LIN {X 0,Y 311.231,Z 437.384,A -85,B 0,C 180,E1 -15755.184,E2 -15755.184} C_VEL
LIN {X 0,Y 311.07,Z 439.493,A -85,B 0,C 180,E1 -15756.488,E2 -15756.488} C_VEL
LIN {X 0,Y 310.876,Z 441.171,A -85,B 0,C 180,E1 -15757.797,E2 -15757.797} C_VEL
LIN {X 0,Y 310.751,Z 442.446,A -85,B 0,C 180,E1 -15759.111,E2 -15759.111} C_VEL
LIN {X 0,Y 310.679,Z 443.314,A -85,B 0,C 180,E1 -15760.428,E2 -15760.428} C_VEL
LIN {X 0,Y 310.751,Z 443.737,A -85,B 0,C 180,E1 -15761.746,E2 -15761.746} C_VEL
LIN {X 0,Y 310.874,Z 443.708,A -85,B 0,C 180,E1 -15763.562,E2 -15763.562} C_VEL
LIN {X 0,Y 311.133,Z 442.642,A -85,B 0,C 180,E1 -15765.728,E2 -15765.728} C_VEL
LIN {X 0,Y 311.417,Z 441.418,A -85,B 0,C 180,E1 -15767.061,E2 -15767.061} C_VEL
LIN {X 0,Y 312.024,Z 439.019,A -85,B 0,C 180,E1 -15768.913,E2 -15768.913} C_VEL
LIN {X 0,Y 312.86,Z 435.083,A -85,B 0,C 180,E1 -15771.065,E2 -15771.065} C_VEL
LIN {X 0,Y 313.883,Z 430.519,A -85,B 0,C 180,E1 -15772.948,E2 -15772.948} C_VEL
LIN {X 0,Y 315.274,Z 423.973,A -85,B 0,C 180,E1 -15775.058,E2 -15775.058} C_VEL
LIN {X 0,Y 316.969,Z 416.151,A -85,B 0,C 180,E1 -15777.035,E2 -15777.035} C_VEL
LIN {X 0,Y 318.681,Z 407.222,A -85,B 0,C 180,E1 -15778.825,E2 -15778.825} C_VEL
LIN {X 0,Y 320.497,Z 396.978,A -85,B 0,C 180,E1 -15780.47,E2 -15780.47} C_VEL
LIN {X 0,Y 322.265,Z 386.498,A -85,B 0,C 180,E1 -15781.793,E2 -15781.793} C_VEL
LIN {X 0,Y 323.658,Z 375.789,A -85,B 0,C 180,E1 -15782.877,E2 -15782.877} C_VEL
LIN {X 0,Y 324.815,Z 364.59,A -85,B 0,C 180,E1 -15783.765,E2 -15783.765} C_VEL
LIN {X 0,Y 325.961,Z 351.288,A -85,B 0,C 180,E1 -15784.526,E2 -15784.526} C_VEL
LIN {X 0,Y 326.606,Z 338.938,A -85,B 0,C 180,E1 -15784.984,E2 -15784.984} C_VEL
LIN {X 0,Y 328.652,Z 266.261,A -85,B 0,C 180,E1 -15786.6,E2 -15786.6} C_VEL
LIN {X 0,Y 321.5,Z 250.026,A -85,B 0,C 180,E1 -15787.749,E2 -15787.749} C_VEL
LIN {X 0,Y 314.331,Z 235.95,A -85,B 0,C 180,E1 -15788.911,E2 -15788.911} C_VEL
LIN {X 0,Y 314.024,Z 235.367,A -85,B 0,C 180,E1 -15788.962,E2 -15788.962} C_VEL
LIN {X 0,Y 312.775,Z 233.899,A -85,B 0,C 180,E1 -15789.216,E2 -15789.216} C_VEL
LIN {X 0,Y 309.925,Z 232.398,A -85,B 0,C 180,E1 -15789.967,E2 -15789.967} C_VEL
LIN {X 0,Y 308.287,Z 231.569,A -85,B 0,C 180,E1 -15790.527,E2 -15790.527} C_VEL
LIN {X 0,Y 306.002,Z 231.431,A -85,B 0,C 180,E1 -15791.683,E2 -15791.683} C_VEL
LIN {X 0,Y 305.488,Z 231.435,A -85,B 0,C 180,E1 -15792.497,E2 -15792.497} C_VEL
LIN {X 0,Y 305.487,Z 231.436,A -85,B 0,C 180,E1 -15796.356,E2 -15796.356} C_VEL
LIN {X 0,Y 305.476,Z 231.431,A -85,B 0,C 180,E1 -15799.895,E2 -15799.895} C_VEL
LIN {X 0,Y 305.474,Z 231.432,A -85,B 0,C 180,E1 -15803.63,E2 -15803.63} C_VEL
LIN {X 0,Y 305.455,Z 231.435,A -85,B 0,C 180,E1 -15806.482,E2 -15806.482} C_VEL
LIN {X 0,Y 305.483,Z 231.432,A -85,B 0,C 180,E1 -15810.95,E2 -15810.95} C_VEL
LIN {X 0,Y 305.557,Z 231.425,A -85,B 0,C 180,E1 -15814.086,E2 -15814.086} C_VEL
LIN {X 0,Y 305.449,Z 231.436,A -85,B 0,C 180,E1 -15818.399,E2 -15818.399} C_VEL
LIN {X 0,Y 305.531,Z 231.419,A -85,B 0,C 180,E1 -15821.214,E2 -15821.214} C_VEL
LIN {X 0,Y 305.608,Z 231.409,A -85,B 0,C 180,E1 -15825.347,E2 -15825.347} C_VEL
LIN {X 0,Y 305.608,Z 231.409,A -85,B 0,C 180,E1 -15829.398,E2 -15829.398} C_VEL
LIN {X 0,Y 305.769,Z 231.395,A -85,B 0,C 180,E1 -15832.073,E2 -15832.073} C_VEL
LIN {X 0,Y 305.662,Z 231.404,A -85,B 0,C 180,E1 -15834.723,E2 -15834.723} C_VEL
LIN {X 0,Y 305.934,Z 231.365,A -85,B 0,C 180,E1 -15838.684,E2 -15838.684} C_VEL
LIN {X 0,Y 305.934,Z 231.375,A -85,B 0,C 180,E1 -15841.316,E2 -15841.316} C_VEL
LIN {X 0,Y 305.648,Z 231.413,A -85,B 0,C 180,E1 -15845.277,E2 -15845.277} C_VEL
LIN {X 0,Y 305.722,Z 231.391,A -85,B 0,C 180,E1 -15847.928,E2 -15847.928} C_VEL
LIN {X 0,Y 305.578,Z 231.412,A -85,B 0,C 180,E1 -15851.946,E2 -15851.946} C_VEL
LIN {X 0,Y 305.591,Z 231.419,A -85,B 0,C 180,E1 -15855.013,E2 -15855.013} C_VEL
LIN {X 0,Y 305.499,Z 231.43,A -85,B 0,C 180,E1 -15858.788,E2 -15858.788} C_VEL
LIN {X 0,Y 305.442,Z 231.438,A -85,B 0,C 180,E1 -15863.027,E2 -15863.027} C_VEL
LIN {X 0,Y 305.438,Z 231.429,A -85,B 0,C 180,E1 -15866.191,E2 -15866.191} C_VEL
LIN {X 0,Y 305.409,Z 231.435,A -85,B 0,C 180,E1 -15869.026,E2 -15869.026} C_VEL
LIN {X 0,Y 305.421,Z 231.44,A -85,B 0,C 180,E1 -15871.955,E2 -15871.955} C_VEL
LIN {X 0,Y 305.449,Z 231.436,A -85,B 0,C 180,E1 -15875.115,E2 -15875.115} C_VEL
LIN {X 0,Y 305.415,Z 231.415,A -85,B 0,C 180,E1 -15878.524,E2 -15878.524} C_VEL
LIN {X 0,Y 305.419,Z 231.442,A -85,B 0,C 180,E1 -15881.861,E2 -15881.861} C_VEL
LIN {X 0,Y 305.392,Z 231.441,A -85,B 0,C 180,E1 -15885.513,E2 -15885.513} C_VEL
LIN {X 0,Y 305.406,Z 231.431,A -85,B 0,C 180,E1 -15888.139,E2 -15888.139} C_VEL
LIN {X 0,Y 305.467,Z 231.429,A -85,B 0,C 180,E1 -15892.434,E2 -15892.434} C_VEL
LIN {X 0,Y 305.527,Z 231.652,A -85,B 0,C 180,E1 -15893.269,E2 -15893.269} C_VEL
LIN {X 0,Y 307.663,Z 239.802,A -85,B 0,C 180,E1 -15896.065,E2 -15896.065} C_VEL
LIN {X 0,Y 310.119,Z 250.307,A -85,B 0,C 180,E1 -15899.448,E2 -15899.448} C_VEL
LIN {X 0,Y 311.704,Z 257.977,A -85,B 0,C 180,E1 -15901.784,E2 -15901.784} C_VEL
LIN {X 0,Y 313.869,Z 263.63,A -85,B 0,C 180,E1 -15902.185,E2 -15902.185} C_VEL
LIN {X 0,Y 318.647,Z 287.185,A -85,B 0,C 180,E1 -15903.318,E2 -15903.318} C_VEL
LIN {X 0,Y 321.489,Z 305.27,A -85,B 0,C 180,E1 -15904.074,E2 -15904.074} C_VEL
LIN {X 0,Y 319.685,Z 367.009,A -85,B 0,C 180,E1 -15905.484,E2 -15905.484} C_VEL
LIN {X 0,Y 318.677,Z 380.224,A -85,B 0,C 180,E1 -15906.008,E2 -15906.008} C_VEL
LIN {X 0,Y 317.293,Z 392.914,A -85,B 0,C 180,E1 -15906.762,E2 -15906.762} C_VEL
LIN {X 0,Y 315.566,Z 405.023,A -85,B 0,C 180,E1 -15907.752,E2 -15907.752} C_VEL
LIN {X 0,Y 313.569,Z 416.536,A -85,B 0,C 180,E1 -15908.985,E2 -15908.985} C_VEL
LIN {X 0,Y 311.699,Z 426.916,A -85,B 0,C 180,E1 -15910.403,E2 -15910.403} C_VEL
LIN {X 0,Y 310.015,Z 435.426,A -85,B 0,C 180,E1 -15911.837,E2 -15911.837} C_VEL
LIN {X 0,Y 308.316,Z 443.862,A -85,B 0,C 180,E1 -15913.578,E2 -15913.578} C_VEL
LIN {X 0,Y 306.923,Z 451.023,A -85,B 0,C 180,E1 -15915.41,E2 -15915.41} C_VEL
LIN {X 0,Y 305.546,Z 457.248,A -85,B 0,C 180,E1 -15917.377,E2 -15917.377} C_VEL
LIN {X 0,Y 304.657,Z 462.223,A -85,B 0,C 180,E1 -15919.364,E2 -15919.364} C_VEL
LIN {X 0,Y 304.066,Z 466.09,A -85,B 0,C 180,E1 -15921.358,E2 -15921.358} C_VEL
LIN {X 0,Y 303.742,Z 468.951,A -85,B 0,C 180,E1 -15923.355,E2 -15923.355} C_VEL
LIN {X 0,Y 303.66,Z 471.296,A -85,B 0,C 180,E1 -15926.016,E2 -15926.016} C_VEL
LIN {X 0,Y 303.656,Z 471.885,A -85,B 0,C 180,E1 -15927.345,E2 -15927.345} C_VEL
LIN {X 0,Y 303.684,Z 472.046,A -85,B 0,C 180,E1 -15928.672,E2 -15928.672} C_VEL
LIN {X 0,Y 303.768,Z 471.804,A -85,B 0,C 180,E1 -15929.998,E2 -15929.998} C_VEL
LIN {X 0,Y 303.723,Z 471.166,A -85,B 0,C 180,E1 -15931.323,E2 -15931.323} C_VEL
LIN {X 0,Y 303.69,Z 470.133,A -85,B 0,C 180,E1 -15932.65,E2 -15932.65} C_VEL
LIN {X 0,Y 303.713,Z 468.654,A -85,B 0,C 180,E1 -15933.978,E2 -15933.978} C_VEL
LIN {X 0,Y 303.728,Z 466.023,A -85,B 0,C 180,E1 -15935.741,E2 -15935.741} C_VEL
LIN {X 0,Y 303.929,Z 461.501,A -85,B 0,C 180,E1 -15937.972,E2 -15937.972} C_VEL
LIN {X 0,Y 304.387,Z 455.17,A -85,B 0,C 180,E1 -15940.304,E2 -15940.304} C_VEL
LIN {X 0,Y 305.062,Z 448.265,A -85,B 0,C 180,E1 -15942.3,E2 -15942.3} C_VEL
LIN {X 0,Y 305.872,Z 441.212,A -85,B 0,C 180,E1 -15943.957,E2 -15943.957} C_VEL
LIN {X 0,Y 306.784,Z 433.425,A -85,B 0,C 180,E1 -15945.476,E2 -15945.476} C_VEL
LIN {X 0,Y 307.98,Z 423.495,A -85,B 0,C 180,E1 -15947.064,E2 -15947.064} C_VEL
LIN {X 0,Y 309.143,Z 413.209,A -85,B 0,C 180,E1 -15948.382,E2 -15948.382} C_VEL
LIN {X 0,Y 310.372,Z 402.142,A -85,B 0,C 180,E1 -15949.507,E2 -15949.507} C_VEL
LIN {X 0,Y 311.519,Z 389.878,A -85,B 0,C 180,E1 -15950.463,E2 -15950.463} C_VEL
LIN {X 0,Y 312.452,Z 377.055,A -85,B 0,C 180,E1 -15951.175,E2 -15951.175} C_VEL
LIN {X 0,Y 313.089,Z 363.48,A -85,B 0,C 180,E1 -15951.648,E2 -15951.648} C_VEL
LIN {X 0,Y 314.139,Z 301.472,A -85,B 0,C 180,E1 -15953.065,E2 -15953.065} C_VEL
LIN {X 0,Y 308.599,Z 258.926,A -85,B 0,C 180,E1 -15954.459,E2 -15954.459} C_VEL
LIN {X 0,Y 309.401,Z 251.713,A -85,B 0,C 180,E1 -15956.286,E2 -15956.286} C_VEL
LIN {X 0,Y 308.464,Z 245.706,A -85,B 0,C 180,E1 -15957.927,E2 -15957.927} C_VEL
LIN {X 0,Y 306.146,Z 234.57,A -85,B 0,C 180,E1 -15961.093,E2 -15961.093} C_VEL
LIN {X 0,Y 305.45,Z 231.442,A -85,B 0,C 180,E1 -15962.042,E2 -15962.042} C_VEL
LIN {X 0,Y 305.444,Z 231.437,A -85,B 0,C 180,E1 -15965.109,E2 -15965.109} C_VEL
LIN {X 0,Y 305.446,Z 231.437,A -85,B 0,C 180,E1 -15968.528,E2 -15968.528} C_VEL
LIN {X 0,Y 305.436,Z 231.437,A -85,B 0,C 180,E1 -15972.582,E2 -15972.582} C_VEL
LIN {X 0,Y 305.461,Z 231.434,A -85,B 0,C 180,E1 -15976.351,E2 -15976.351} C_VEL
LIN {X 0,Y 305.455,Z 231.438,A -85,B 0,C 180,E1 -15979.892,E2 -15979.892} C_VEL
LIN {X 0,Y 305.468,Z 231.436,A -85,B 0,C 180,E1 -15983.623,E2 -15983.623} C_VEL
LIN {X 0,Y 305.432,Z 231.436,A -85,B 0,C 180,E1 -15986.479,E2 -15986.479} C_VEL
LIN {X 0,Y 305.459,Z 231.434,A -85,B 0,C 180,E1 -15990.947,E2 -15990.947} C_VEL
LIN {X 0,Y 305.535,Z 231.424,A -85,B 0,C 180,E1 -15994.085,E2 -15994.085} C_VEL
LIN {X 0,Y 305.519,Z 231.425,A -85,B 0,C 180,E1 -15998.404,E2 -15998.404} C_VEL
LIN {X 0,Y 305.552,Z 231.425,A -85,B 0,C 180,E1 -16001.215,E2 -16001.215} C_VEL
LIN {X 0,Y 305.595,Z 231.419,A -85,B 0,C 180,E1 -16005.346,E2 -16005.346} C_VEL
LIN {X 0,Y 305.595,Z 231.42,A -85,B 0,C 180,E1 -16009.398,E2 -16009.398} C_VEL
LIN {X 0,Y 305.766,Z 231.393,A -85,B 0,C 180,E1 -16012.073,E2 -16012.073} C_VEL
LIN {X 0,Y 305.647,Z 231.411,A -85,B 0,C 180,E1 -16014.723,E2 -16014.723} C_VEL
LIN {X 0,Y 305.911,Z 231.377,A -85,B 0,C 180,E1 -16018.684,E2 -16018.684} C_VEL
LIN {X 0,Y 305.91,Z 231.37,A -85,B 0,C 180,E1 -16021.317,E2 -16021.317} C_VEL
LIN {X 0,Y 305.793,Z 231.392,A -85,B 0,C 180,E1 -16026.599,E2 -16026.599} C_VEL
LIN {X 0,Y 305.656,Z 231.41,A -85,B 0,C 180,E1 -16029.262,E2 -16029.262} C_VEL
LIN {X 0,Y 305.542,Z 231.416,A -85,B 0,C 180,E1 -16033.298,E2 -16033.298} C_VEL
LIN {X 0,Y 305.511,Z 231.421,A -85,B 0,C 180,E1 -16036.025,E2 -16036.025} C_VEL
LIN {X 0,Y 305.441,Z 231.436,A -85,B 0,C 180,E1 -16040.191,E2 -16040.191} C_VEL
LIN {X 0,Y 305.466,Z 231.434,A -85,B 0,C 180,E1 -16044.465,E2 -16044.465} C_VEL
LIN {X 0,Y 305.463,Z 231.432,A -85,B 0,C 180,E1 -16047.397,E2 -16047.397} C_VEL
LIN {X 0,Y 305.428,Z 231.44,A -85,B 0,C 180,E1 -16050.413,E2 -16050.413} C_VEL
LIN {X 0,Y 305.432,Z 231.438,A -85,B 0,C 180,E1 -16054.082,E2 -16054.082} C_VEL
LIN {X 0,Y 305.466,Z 231.434,A -85,B 0,C 180,E1 -16056.741,E2 -16056.741} C_VEL
LIN {X 0,Y 305.457,Z 231.436,A -85,B 0,C 180,E1 -16060.611,E2 -16060.611} C_VEL
LIN {X 0,Y 305.462,Z 231.432,A -85,B 0,C 180,E1 -16063.649,E2 -16063.649} C_VEL
LIN {X 0,Y 305.437,Z 231.433,A -85,B 0,C 180,E1 -16067.418,E2 -16067.418} C_VEL
LIN {X 0,Y 305.448,Z 231.434,A -85,B 0,C 180,E1 -16071.601,E2 -16071.601} C_VEL
LIN {X 0,Y 305.445,Z 231.434,A -85,B 0,C 180,E1 -16074.892,E2 -16074.892} C_VEL
LIN {X 0,Y 305.436,Z 231.438,A -85,B 0,C 180,E1 -16078.361,E2 -16078.361} C_VEL
LIN {X 0,Y 305.501,Z 231.428,A -85,B 0,C 180,E1 -16081.118,E2 -16081.118} C_VEL
LIN {X 0,Y 305.561,Z 231.423,A -85,B 0,C 180,E1 -16084.092,E2 -16084.092} C_VEL
LIN {X 0,Y 305.467,Z 231.433,A -85,B 0,C 180,E1 -16088.405,E2 -16088.405} C_VEL
LIN {X 0,Y 305.512,Z 231.428,A -85,B 0,C 180,E1 -16091.217,E2 -16091.217} C_VEL
LIN {X 0,Y 305.653,Z 231.413,A -85,B 0,C 180,E1 -16095.693,E2 -16095.693} C_VEL
LIN {X 0,Y 305.679,Z 231.523,A -85,B 0,C 180,E1 -16095.949,E2 -16095.949} C_VEL
LIN {X 0,Y 306.071,Z 233.404,A -85,B 0,C 180,E1 -16096.46,E2 -16096.46} C_VEL
LIN {X 0,Y 314.005,Z 256.117,A -85,B 0,C 180,E1 -16097.562,E2 -16097.562} C_VEL
LIN {X 0,Y 314.979,Z 263.205,A -85,B 0,C 180,E1 -16097.796,E2 -16097.796} C_VEL
LIN {X 0,Y 313.197,Z 339.943,A -85,B 0,C 180,E1 -16099.539,E2 -16099.539} C_VEL
LIN {X 0,Y 312.519,Z 353.304,A -85,B 0,C 180,E1 -16100.089,E2 -16100.089} C_VEL
LIN {X 0,Y 311.82,Z 365.425,A -85,B 0,C 180,E1 -16100.844,E2 -16100.844} C_VEL
LIN {X 0,Y 311.13,Z 375.954,A -85,B 0,C 180,E1 -16101.724,E2 -16101.724} C_VEL
LIN {X 0,Y 309.996,Z 386.647,A -85,B 0,C 180,E1 -16102.84,E2 -16102.84} C_VEL
LIN {X 0,Y 308.887,Z 396.47,A -85,B 0,C 180,E1 -16104.126,E2 -16104.126} C_VEL
LIN {X 0,Y 307.67,Z 406.407,A -85,B 0,C 180,E1 -16105.745,E2 -16105.745} C_VEL
LIN {X 0,Y 306.558,Z 416.019,A -85,B 0,C 180,E1 -16107.703,E2 -16107.703} C_VEL
LIN {X 0,Y 305.502,Z 423.71,A -85,B 0,C 180,E1 -16109.673,E2 -16109.673} C_VEL
LIN {X 0,Y 304.806,Z 430.761,A -85,B 0,C 180,E1 -16111.984,E2 -16111.984} C_VEL
LIN {X 0,Y 304.267,Z 435.478,A -85,B 0,C 180,E1 -16113.976,E2 -16113.976} C_VEL
LIN {X 0,Y 304.02,Z 439.536,A -85,B 0,C 180,E1 -16116.262,E2 -16116.262} C_VEL
LIN {X 0,Y 303.767,Z 441.688,A -85,B 0,C 180,E1 -16117.981,E2 -16117.981} C_VEL
LIN {X 0,Y 303.635,Z 442.921,A -85,B 0,C 180,E1 -16119.326,E2 -16119.326} C_VEL
LIN {X 0,Y 303.588,Z 443.709,A -85,B 0,C 180,E1 -16120.674,E2 -16120.674} C_VEL
LIN {X 0,Y 303.678,Z 444.089,A -85,B 0,C 180,E1 -16122.023,E2 -16122.023} C_VEL
LIN {X 0,Y 303.81,Z 444.042,A -85,B 0,C 180,E1 -16123.69,E2 -16123.69} C_VEL
LIN {X 0,Y 304.122,Z 442.829,A -85,B 0,C 180,E1 -16126.101,E2 -16126.101} C_VEL
LIN {X 0,Y 304.461,Z 441.563,A -85,B 0,C 180,E1 -16127.464,E2 -16127.464} C_VEL
LIN {X 0,Y 305.041,Z 439.395,A -85,B 0,C 180,E1 -16129.156,E2 -16129.156} C_VEL
LIN {X 0,Y 306.014,Z 435.046,A -85,B 0,C 180,E1 -16131.56,E2 -16131.56} C_VEL
LIN {X 0,Y 307.334,Z 429.428,A -85,B 0,C 180,E1 -16133.835,E2 -16133.835} C_VEL
LIN {X 0,Y 308.93,Z 422.498,A -85,B 0,C 180,E1 -16135.972,E2 -16135.972} C_VEL
LIN {X 0,Y 310.695,Z 414.327,A -85,B 0,C 180,E1 -16137.959,E2 -16137.959} C_VEL
LIN {X 0,Y 312.444,Z 405.615,A -85,B 0,C 180,E1 -16139.66,E2 -16139.66} C_VEL
LIN {X 0,Y 314.367,Z 395.151,A -85,B 0,C 180,E1 -16141.283,E2 -16141.283} C_VEL
LIN {X 0,Y 316.199,Z 384.268,A -85,B 0,C 180,E1 -16142.614,E2 -16142.614} C_VEL
LIN {X 0,Y 317.715,Z 372.402,A -85,B 0,C 180,E1 -16143.763,E2 -16143.763} C_VEL
LIN {X 0,Y 318.898,Z 361.267,A -85,B 0,C 180,E1 -16144.574,E2 -16144.574} C_VEL
LIN {X 0,Y 319.89,Z 347.987,A -85,B 0,C 180,E1 -16145.269,E2 -16145.269} C_VEL
LIN {X 0,Y 320.547,Z 334.719,A -85,B 0,C 180,E1 -16145.691,E2 -16145.691} C_VEL
LIN {X 0,Y 322.434,Z 268.162,A -85,B 0,C 180,E1 -16147.186,E2 -16147.186} C_VEL
LIN {X 0,Y 315.594,Z 252.633,A -85,B 0,C 180,E1 -16148.327,E2 -16148.327} C_VEL
LIN {X 0,Y 307.919,Z 237.531,A -85,B 0,C 180,E1 -16149.625,E2 -16149.625} C_VEL
LIN {X 0,Y 306.139,Z 234.045,A -85,B 0,C 180,E1 -16149.958,E2 -16149.958} C_VEL
LIN {X 0,Y 305.451,Z 231.434,A -85,B 0,C 180,E1 -16150.997,E2 -16150.997} C_VEL
LIN {X 0,Y 305.488,Z 231.435,A -85,B 0,C 180,E1 -16152.497,E2 -16152.497} C_VEL
LIN {X 0,Y 304.853,Z 231.512,A -85,B 0,C 180,E1 -16153.596,E2 -16153.596} C_VEL
LIN {X 0,Y 301.975,Z 231.868,A -85,B 0,C 180,E1 -16155.383,E2 -16155.383} C_VEL
LIN {X 0,Y 299.525,Z 232.176,A -85,B 0,C 180,E1 -16156.834,E2 -16156.834} C_VEL
LIN {X 0,Y 298.494,Z 232.303,A -85,B 0,C 180,E1 -16157.958,E2 -16157.958} C_VEL
LIN {X 0,Y 298.423,Z 232.31,A -85,B 0,C 180,E1 -16158.339,E2 -16158.339} C_VEL
LIN {X 0,Y 298.426,Z 232.307,A -85,B 0,C 180,E1 -16162.243,E2 -16162.243} C_VEL
LIN {X 0,Y 298.398,Z 232.31,A -85,B 0,C 180,E1 -16165.579,E2 -16165.579} C_VEL
LIN {X 0,Y 298.383,Z 232.31,A -85,B 0,C 180,E1 -16168.789,E2 -16168.789} C_VEL
LIN {X 0,Y 298.45,Z 232.303,A -85,B 0,C 180,E1 -16171.903,E2 -16171.903} C_VEL
LIN {X 0,Y 298.47,Z 232.305,A -85,B 0,C 180,E1 -16174.922,E2 -16174.922} C_VEL
LIN {X 0,Y 298.41,Z 232.311,A -85,B 0,C 180,E1 -16179.312,E2 -16179.312} C_VEL
LIN {X 0,Y 298.495,Z 232.303,A -85,B 0,C 180,E1 -16182.177,E2 -16182.177} C_VEL
LIN {X 0,Y 298.572,Z 232.283,A -85,B 0,C 180,E1 -16184.993,E2 -16184.993} C_VEL
LIN {X 0,Y 298.567,Z 232.285,A -85,B 0,C 180,E1 -16189.145,E2 -16189.145} C_VEL
LIN {X 0,Y 298.715,Z 232.274,A -85,B 0,C 180,E1 -16191.885,E2 -16191.885} C_VEL
LIN {X 0,Y 298.634,Z 232.279,A -85,B 0,C 180,E1 -16194.598,E2 -16194.598} C_VEL
LIN {X 0,Y 298.901,Z 232.241,A -85,B 0,C 180,E1 -16198.653,E2 -16198.653} C_VEL
LIN {X 0,Y 298.9,Z 232.25,A -85,B 0,C 180,E1 -16201.347,E2 -16201.347} C_VEL
LIN {X 0,Y 298.617,Z 232.288,A -85,B 0,C 180,E1 -16205.402,E2 -16205.402} C_VEL
LIN {X 0,Y 298.668,Z 232.27,A -85,B 0,C 180,E1 -16208.116,E2 -16208.116} C_VEL
LIN {X 0,Y 298.53,Z 232.288,A -85,B 0,C 180,E1 -16212.232,E2 -16212.232} C_VEL
LIN {X 0,Y 298.53,Z 232.297,A -85,B 0,C 180,E1 -16215.166,E2 -16215.166} C_VEL
LIN {X 0,Y 298.423,Z 232.31,A -85,B 0,C 180,E1 -16219.615,E2 -16219.615} C_VEL
LIN {X 0,Y 298.374,Z 232.317,A -85,B 0,C 180,E1 -16223.605,E2 -16223.605} C_VEL
LIN {X 0,Y 298.389,Z 232.31,A -85,B 0,C 180,E1 -16226.584,E2 -16226.584} C_VEL
LIN {X 0,Y 298.342,Z 232.313,A -85,B 0,C 180,E1 -16229.65,E2 -16229.65} C_VEL
LIN {X 0,Y 298.379,Z 232.311,A -85,B 0,C 180,E1 -16232.802,E2 -16232.802} C_VEL
LIN {X 0,Y 298.393,Z 232.313,A -85,B 0,C 180,E1 -16236.073,E2 -16236.073} C_VEL
LIN {X 0,Y 298.387,Z 232.295,A -85,B 0,C 180,E1 -16239.49,E2 -16239.49} C_VEL
LIN {X 0,Y 298.393,Z 232.313,A -85,B 0,C 180,E1 -16243.104,E2 -16243.104} C_VEL
LIN {X 0,Y 298.364,Z 232.318,A -85,B 0,C 180,E1 -16246.916,E2 -16246.916} C_VEL
LIN {X 0,Y 298.381,Z 232.312,A -85,B 0,C 180,E1 -16251.012,E2 -16251.012} C_VEL
LIN {X 0,Y 298.439,Z 232.36,A -85,B 0,C 180,E1 -16252.447,E2 -16252.447} C_VEL
LIN {X 0,Y 301.01,Z 242.169,A -85,B 0,C 180,E1 -16255.921,E2 -16255.921} C_VEL
LIN {X 0,Y 303.439,Z 252.629,A -85,B 0,C 180,E1 -16259.367,E2 -16259.367} C_VEL
LIN {X 0,Y 304.525,Z 257.639,A -85,B 0,C 180,E1 -16260.932,E2 -16260.932} C_VEL
LIN {X 0,Y 308.152,Z 266.663,A -85,B 0,C 180,E1 -16261.612,E2 -16261.612} C_VEL
LIN {X 0,Y 312.66,Z 289.196,A -85,B 0,C 180,E1 -16262.726,E2 -16262.726} C_VEL
LIN {X 0,Y 315.3,Z 305.796,A -85,B 0,C 180,E1 -16263.446,E2 -16263.446} C_VEL
LIN {X 0,Y 313.446,Z 366.947,A -85,B 0,C 180,E1 -16264.874,E2 -16264.874} C_VEL
LIN {X 0,Y 312.323,Z 380.823,A -85,B 0,C 180,E1 -16265.443,E2 -16265.443} C_VEL
LIN {X 0,Y 310.818,Z 393.79,A -85,B 0,C 180,E1 -16266.249,E2 -16266.249} C_VEL
LIN {X 0,Y 309.048,Z 405.56,A -85,B 0,C 180,E1 -16267.257,E2 -16267.257} C_VEL
LIN {X 0,Y 306.978,Z 416.911,A -85,B 0,C 180,E1 -16268.512,E2 -16268.512} C_VEL
LIN {X 0,Y 305.04,Z 427.163,A -85,B 0,C 180,E1 -16269.957,E2 -16269.957} C_VEL
LIN {X 0,Y 302.885,Z 437.219,A -85,B 0,C 180,E1 -16271.744,E2 -16271.744} C_VEL
LIN {X 0,Y 301.03,Z 446.079,A -85,B 0,C 180,E1 -16273.729,E2 -16273.729} C_VEL
LIN {X 0,Y 299.506,Z 453.228,A -85,B 0,C 180,E1 -16275.735,E2 -16275.735} C_VEL
LIN {X 0,Y 298.195,Z 458.956,A -85,B 0,C 180,E1 -16277.752,E2 -16277.752} C_VEL
LIN {X 0,Y 297.404,Z 463.498,A -85,B 0,C 180,E1 -16279.79,E2 -16279.79} C_VEL
LIN {X 0,Y 296.882,Z 466.974,A -85,B 0,C 180,E1 -16281.833,E2 -16281.833} C_VEL
LIN {X 0,Y 296.553,Z 470.065,A -85,B 0,C 180,E1 -16284.558,E2 -16284.558} C_VEL
LIN {X 0,Y 296.573,Z 471.022,A -85,B 0,C 180,E1 -16285.921,E2 -16285.921} C_VEL
LIN {X 0,Y 296.579,Z 471.581,A -85,B 0,C 180,E1 -16287.281,E2 -16287.281} C_VEL
LIN {X 0,Y 296.596,Z 471.707,A -85,B 0,C 180,E1 -16288.64,E2 -16288.64} C_VEL
LIN {X 0,Y 296.676,Z 471.444,A -85,B 0,C 180,E1 -16289.997,E2 -16289.997} C_VEL
LIN {X 0,Y 296.634,Z 470.785,A -85,B 0,C 180,E1 -16291.355,E2 -16291.355} C_VEL
LIN {X 0,Y 296.613,Z 469.726,A -85,B 0,C 180,E1 -16292.713,E2 -16292.713} C_VEL
LIN {X 0,Y 296.625,Z 468.206,A -85,B 0,C 180,E1 -16294.073,E2 -16294.073} C_VEL
LIN {X 0,Y 296.675,Z 465.122,A -85,B 0,C 180,E1 -16296.116,E2 -16296.116} C_VEL
LIN {X 0,Y 296.86,Z 460.953,A -85,B 0,C 180,E1 -16298.163,E2 -16298.163} C_VEL
LIN {X 0,Y 297.348,Z 454.564,A -85,B 0,C 180,E1 -16300.551,E2 -16300.551} C_VEL
LIN {X 0,Y 298.107,Z 447.601,A -85,B 0,C 180,E1 -16302.592,E2 -16302.592} C_VEL
LIN {X 0,Y 298.924,Z 440.475,A -85,B 0,C 180,E1 -16304.288,E2 -16304.288} C_VEL
LIN {X 0,Y 299.894,Z 432.13,A -85,B 0,C 180,E1 -16305.93,E2 -16305.93} C_VEL
LIN {X 0,Y 301.142,Z 422.401,A -85,B 0,C 180,E1 -16307.482,E2 -16307.482} C_VEL
LIN {X 0,Y 302.329,Z 412.091,A -85,B 0,C 180,E1 -16308.812,E2 -16308.812} C_VEL
LIN {X 0,Y 303.631,Z 400.841,A -85,B 0,C 180,E1 -16309.958,E2 -16309.958} C_VEL
LIN {X 0,Y 304.828,Z 388.233,A -85,B 0,C 180,E1 -16310.933,E2 -16310.933} C_VEL
LIN {X 0,Y 305.755,Z 375.643,A -85,B 0,C 180,E1 -16311.618,E2 -16311.618} C_VEL
LIN {X 0,Y 306.354,Z 362.88,A -85,B 0,C 180,E1 -16312.06,E2 -16312.06} C_VEL
LIN {X 0,Y 307.445,Z 302.149,A -85,B 0,C 180,E1 -16313.476,E2 -16313.476} C_VEL
LIN {X 0,Y 301.907,Z 259.709,A -85,B 0,C 180,E1 -16314.903,E2 -16314.903} C_VEL
LIN {X 0,Y 301.766,Z 258.54,A -85,B 0,C 180,E1 -16314.961,E2 -16314.961} C_VEL
LIN {X 0,Y 302.425,Z 252.358,A -85,B 0,C 180,E1 -16316.568,E2 -16316.568} C_VEL
LIN {X 0,Y 300.595,Z 242.377,A -85,B 0,C 180,E1 -16319.399,E2 -16319.399} C_VEL
LIN {X 0,Y 298.424,Z 232.316,A -85,B 0,C 180,E1 -16322.401,E2 -16322.401} C_VEL
LIN {X 0,Y 298.4,Z 232.318,A -85,B 0,C 180,E1 -16326.065,E2 -16326.065} C_VEL
LIN {X 0,Y 298.388,Z 232.317,A -85,B 0,C 180,E1 -16329.482,E2 -16329.482} C_VEL
LIN {X 0,Y 298.376,Z 232.316,A -85,B 0,C 180,E1 -16333.099,E2 -16333.099} C_VEL
LIN {X 0,Y 298.414,Z 232.311,A -85,B 0,C 180,E1 -16336.923,E2 -16336.923} C_VEL
LIN {X 0,Y 298.398,Z 232.313,A -85,B 0,C 180,E1 -16340.512,E2 -16340.512} C_VEL
LIN {X 0,Y 298.4,Z 232.316,A -85,B 0,C 180,E1 -16343.928,E2 -16343.928} C_VEL
LIN {X 0,Y 298.361,Z 232.32,A -85,B 0,C 180,E1 -16347.98,E2 -16347.98} C_VEL
LIN {X 0,Y 298.427,Z 232.311,A -85,B 0,C 180,E1 -16351.901,E2 -16351.901} C_VEL
LIN {X 0,Y 298.461,Z 232.306,A -85,B 0,C 180,E1 -16354.922,E2 -16354.922} C_VEL
LIN {X 0,Y 298.452,Z 232.307,A -85,B 0,C 180,E1 -16357.866,E2 -16357.866} C_VEL
LIN {X 0,Y 298.519,Z 232.298,A -85,B 0,C 180,E1 -16360.756,E2 -16360.756} C_VEL
LIN {X 0,Y 298.546,Z 232.297,A -85,B 0,C 180,E1 -16364.992,E2 -16364.992} C_VEL
LIN {X 0,Y 298.551,Z 232.297,A -85,B 0,C 180,E1 -16369.145,E2 -16369.145} C_VEL
LIN {X 0,Y 298.712,Z 232.272,A -85,B 0,C 180,E1 -16371.885,E2 -16371.885} C_VEL
LIN {X 0,Y 298.618,Z 232.285,A -85,B 0,C 180,E1 -16374.598,E2 -16374.598} C_VEL
LIN {X 0,Y 298.878,Z 232.253,A -85,B 0,C 180,E1 -16378.653,E2 -16378.653} C_VEL
LIN {X 0,Y 298.877,Z 232.244,A -85,B 0,C 180,E1 -16381.348,E2 -16381.348} C_VEL
LIN {X 0,Y 298.738,Z 232.272,A -85,B 0,C 180,E1 -16386.755,E2 -16386.755} C_VEL
LIN {X 0,Y 298.588,Z 232.289,A -85,B 0,C 180,E1 -16389.484,E2 -16389.484} C_VEL
LIN {X 0,Y 298.501,Z 232.291,A -85,B 0,C 180,E1 -16393.618,E2 -16393.618} C_VEL
LIN {X 0,Y 298.445,Z 232.302,A -85,B 0,C 180,E1 -16396.415,E2 -16396.415} C_VEL
LIN {X 0,Y 298.404,Z 232.312,A -85,B 0,C 180,E1 -16399.62,E2 -16399.62} C_VEL
LIN {X 0,Y 298.392,Z 232.311,A -85,B 0,C 180,E1 -16403.603,E2 -16403.603} C_VEL
LIN {X 0,Y 298.449,Z 232.311,A -85,B 0,C 180,E1 -16406.579,E2 -16406.579} C_VEL
LIN {X 0,Y 298.386,Z 232.313,A -85,B 0,C 180,E1 -16409.645,E2 -16409.645} C_VEL
LIN {X 0,Y 298.363,Z 232.318,A -85,B 0,C 180,E1 -16412.805,E2 -16412.805} C_VEL
LIN {X 0,Y 298.435,Z 232.31,A -85,B 0,C 180,E1 -16416.816,E2 -16416.816} C_VEL
LIN {X 0,Y 298.425,Z 232.309,A -85,B 0,C 180,E1 -16421.255,E2 -16421.255} C_VEL
LIN {X 0,Y 298.366,Z 232.311,A -85,B 0,C 180,E1 -16424.963,E2 -16424.963} C_VEL
LIN {X 0,Y 298.367,Z 232.316,A -85,B 0,C 180,E1 -16428.917,E2 -16428.917} C_VEL
LIN {X 0,Y 298.426,Z 232.305,A -85,B 0,C 180,E1 -16433.198,E2 -16433.198} C_VEL
LIN {X 0,Y 298.38,Z 232.314,A -85,B 0,C 180,E1 -16437.205,E2 -16437.205} C_VEL
LIN {X 0,Y 298.415,Z 232.312,A -85,B 0,C 180,E1 -16440.621,E2 -16440.621} C_VEL
LIN {X 0,Y 298.472,Z 232.305,A -85,B 0,C 180,E1 -16443.48,E2 -16443.48} C_VEL
LIN {X 0,Y 298.423,Z 232.309,A -85,B 0,C 180,E1 -16446.704,E2 -16446.704} C_VEL
LIN {X 0,Y 298.472,Z 232.304,A -85,B 0,C 180,E1 -16450.757,E2 -16450.757} C_VEL
LIN {X 0,Y 298.647,Z 232.451,A -85,B 0,C 180,E1 -16455.612,E2 -16455.612} C_VEL
LIN {X 0,Y 298.895,Z 233.68,A -85,B 0,C 180,E1 -16455.94,E2 -16455.94} C_VEL
LIN {X 0,Y 307.238,Z 257.186,A -85,B 0,C 180,E1 -16457.129,E2 -16457.129} C_VEL
LIN {X 0,Y 308.34,Z 262.859,A -85,B 0,C 180,E1 -16457.344,E2 -16457.344} C_VEL
LIN {X 0,Y 306.45,Z 340.325,A -85,B 0,C 180,E1 -16459.139,E2 -16459.139} C_VEL
LIN {X 0,Y 305.754,Z 353.661,A -85,B 0,C 180,E1 -16459.7,E2 -16459.7} C_VEL
LIN {X 0,Y 305.028,Z 365.773,A -85,B 0,C 180,E1 -16460.471,E2 -16460.471} C_VEL
LIN {X 0,Y 304.307,Z 376.297,A -85,B 0,C 180,E1 -16461.37,E2 -16461.37} C_VEL
LIN {X 0,Y 303.139,Z 386.985,A -85,B 0,C 180,E1 -16462.51,E2 -16462.51} C_VEL
LIN {X 0,Y 301.992,Z 396.805,A -85,B 0,C 180,E1 -16463.824,E2 -16463.824} C_VEL
LIN {X 0,Y 300.856,Z 405.852,A -85,B 0,C 180,E1 -16465.313,E2 -16465.313} C_VEL
LIN {X 0,Y 299.824,Z 414.137,A -85,B 0,C 180,E1 -16466.98,E2 -16466.98} C_VEL
LIN {X 0,Y 298.769,Z 422.255,A -85,B 0,C 180,E1 -16468.992,E2 -16468.992} C_VEL
LIN {X 0,Y 298.024,Z 427.793,A -85,B 0,C 180,E1 -16470.678,E2 -16470.678} C_VEL
LIN {X 0,Y 297.54,Z 433.187,A -85,B 0,C 180,E1 -16472.71,E2 -16472.71} C_VEL
LIN {X 0,Y 297.121,Z 437.424,A -85,B 0,C 180,E1 -16474.751,E2 -16474.751} C_VEL
LIN {X 0,Y 296.837,Z 440.607,A -85,B 0,C 180,E1 -16476.801,E2 -16476.801} C_VEL
LIN {X 0,Y 296.652,Z 442.202,A -85,B 0,C 180,E1 -16478.174,E2 -16478.174} C_VEL
LIN {X 0,Y 296.529,Z 443.369,A -85,B 0,C 180,E1 -16479.552,E2 -16479.552} C_VEL
LIN {X 0,Y 296.596,Z 444.441,A -85,B 0,C 180,E1 -16482.315,E2 -16482.315} C_VEL
LIN {X 0,Y 296.744,Z 444.377,A -85,B 0,C 180,E1 -16483.823,E2 -16483.823} C_VEL
LIN {X 0,Y 297.125,Z 443.017,A -85,B 0,C 180,E1 -16486.491,E2 -16486.491} C_VEL
LIN {X 0,Y 297.501,Z 441.708,A -85,B 0,C 180,E1 -16487.886,E2 -16487.886} C_VEL
LIN {X 0,Y 298.218,Z 439.006,A -85,B 0,C 180,E1 -16489.91,E2 -16489.91} C_VEL
LIN {X 0,Y 299.193,Z 435.01,A -85,B 0,C 180,E1 -16492.077,E2 -16492.077} C_VEL
LIN {X 0,Y 300.474,Z 429.859,A -85,B 0,C 180,E1 -16494.188,E2 -16494.188} C_VEL
LIN {X 0,Y 302.056,Z 423.448,A -85,B 0,C 180,E1 -16496.236,E2 -16496.236} C_VEL
LIN {X 0,Y 303.758,Z 416.047,A -85,B 0,C 180,E1 -16498.121,E2 -16498.121} C_VEL
LIN {X 0,Y 305.705,Z 406.854,A -85,B 0,C 180,E1 -16500.001,E2 -16500.001} C_VEL
LIN {X 0,Y 307.719,Z 396.465,A -85,B 0,C 180,E1 -16501.688,E2 -16501.688} C_VEL
LIN {X 0,Y 309.599,Z 386.073,A -85,B 0,C 180,E1 -16503.011,E2 -16503.011} C_VEL
LIN {X 0,Y 311.144,Z 374.604,A -85,B 0,C 180,E1 -16504.184,E2 -16504.184} C_VEL
LIN {X 0,Y 312.335,Z 364.074,A -85,B 0,C 180,E1 -16505.014,E2 -16505.014} C_VEL
LIN {X 0,Y 313.508,Z 351.168,A -85,B 0,C 180,E1 -16505.753,E2 -16505.753} C_VEL
LIN {X 0,Y 314.195,Z 338.728,A -85,B 0,C 180,E1 -16506.214,E2 -16506.214} C_VEL
LIN {X 0,Y 316.311,Z 270.212,A -85,B 0,C 180,E1 -16507.787,E2 -16507.787} C_VEL
LIN {X 0,Y 309.711,Z 255.238,A -85,B 0,C 180,E1 -16508.929,E2 -16508.929} C_VEL
LIN {X 0,Y 301.837,Z 239.963,A -85,B 0,C 180,E1 -16510.31,E2 -16510.31} C_VEL
LIN {X 0,Y 298.959,Z 234.434,A -85,B 0,C 180,E1 -16510.86,E2 -16510.86} C_VEL
LIN {X 0,Y 298.424,Z 232.317,A -85,B 0,C 180,E1 -16511.704,E2 -16511.704} C_VEL
LIN {X 0,Y 298.413,Z 232.308,A -85,B 0,C 180,E1 -16515.046,E2 -16515.046} C_VEL
LIN {X 0,Y 298.423,Z 232.31,A -85,B 0,C 180,E1 -16518.339,E2 -16518.339} C_VEL
LIN {X 0,Y 297.782,Z 232.395,A -85,B 0,C 180,E1 -16519.465,E2 -16519.465} C_VEL
LIN {X 0,Y 294.908,Z 232.751,A -85,B 0,C 180,E1 -16521.297,E2 -16521.297} C_VEL
LIN {X 0,Y 292.46,Z 233.049,A -85,B 0,C 180,E1 -16522.784,E2 -16522.784} C_VEL
LIN {X 0,Y 291.422,Z 233.185,A -85,B 0,C 180,E1 -16523.936,E2 -16523.936} C_VEL
LIN {X 0,Y 291.345,Z 233.19,A -85,B 0,C 180,E1 -16524.327,E2 -16524.327} C_VEL
LIN {X 0,Y 291.361,Z 233.19,A -85,B 0,C 180,E1 -16527.949,E2 -16527.949} C_VEL
LIN {X 0,Y 291.37,Z 233.191,A -85,B 0,C 180,E1 -16531.157,E2 -16531.157} C_VEL
LIN {X 0,Y 291.401,Z 233.187,A -85,B 0,C 180,E1 -16534.27,E2 -16534.27} C_VEL
LIN {X 0,Y 291.356,Z 233.186,A -85,B 0,C 180,E1 -16537.297,E2 -16537.297} C_VEL
LIN {X 0,Y 291.427,Z 233.173,A -85,B 0,C 180,E1 -16540.268,E2 -16540.268} C_VEL
LIN {X 0,Y 291.484,Z 233.166,A -85,B 0,C 180,E1 -16544.665,E2 -16544.665} C_VEL
LIN {X 0,Y 291.512,Z 233.164,A -85,B 0,C 180,E1 -16548.879,E2 -16548.879} C_VEL
LIN {X 0,Y 291.663,Z 233.154,A -85,B 0,C 180,E1 -16551.687,E2 -16551.687} C_VEL
LIN {X 0,Y 291.605,Z 233.155,A -85,B 0,C 180,E1 -16554.468,E2 -16554.468} C_VEL
LIN {X 0,Y 291.867,Z 233.117,A -85,B 0,C 180,E1 -16558.62,E2 -16558.62} C_VEL
LIN {X 0,Y 291.867,Z 233.126,A -85,B 0,C 180,E1 -16561.38,E2 -16561.38} C_VEL
LIN {X 0,Y 291.668,Z 233.145,A -85,B 0,C 180,E1 -16566.92,E2 -16566.92} C_VEL
LIN {X 0,Y 291.546,Z 233.167,A -85,B 0,C 180,E1 -16569.715,E2 -16569.715} C_VEL
LIN {X 0,Y 291.497,Z 233.171,A -85,B 0,C 180,E1 -16573.951,E2 -16573.951} C_VEL
LIN {X 0,Y 291.411,Z 233.176,A -85,B 0,C 180,E1 -16576.822,E2 -16576.822} C_VEL
LIN {X 0,Y 291.378,Z 233.188,A -85,B 0,C 180,E1 -16579.843,E2 -16579.843} C_VEL
LIN {X 0,Y 291.319,Z 233.198,A -85,B 0,C 180,E1 -16584.212,E2 -16584.212} C_VEL
LIN {X 0,Y 291.316,Z 233.198,A -85,B 0,C 180,E1 -16587.282,E2 -16587.282} C_VEL
LIN {X 0,Y 291.287,Z 233.194,A -85,B 0,C 180,E1 -16590.443,E2 -16590.443} C_VEL
LIN {X 0,Y 291.331,Z 233.186,A -85,B 0,C 180,E1 -16593.7,E2 -16593.7} C_VEL
LIN {X 0,Y 291.346,Z 233.175,A -85,B 0,C 180,E1 -16597.249,E2 -16597.249} C_VEL
LIN {X 0,Y 291.319,Z 233.191,A -85,B 0,C 180,E1 -16600.645,E2 -16600.645} C_VEL
LIN {X 0,Y 291.285,Z 233.201,A -85,B 0,C 180,E1 -16604.403,E2 -16604.403} C_VEL
LIN {X 0,Y 291.289,Z 233.188,A -85,B 0,C 180,E1 -16608.413,E2 -16608.413} C_VEL
LIN {X 0,Y 291.38,Z 233.363,A -85,B 0,C 180,E1 -16611.679,E2 -16611.679} C_VEL
LIN {X 0,Y 294.15,Z 243.558,A -85,B 0,C 180,E1 -16615.429,E2 -16615.429} C_VEL
LIN {X 0,Y 296.523,Z 253.911,A -85,B 0,C 180,E1 -16618.94,E2 -16618.94} C_VEL
LIN {X 0,Y 297.236,Z 257.231,A -85,B 0,C 180,E1 -16620.008,E2 -16620.008} C_VEL
LIN {X 0,Y 302.364,Z 269.064,A -85,B 0,C 180,E1 -16620.986,E2 -16620.986} C_VEL
LIN {X 0,Y 306.69,Z 290.958,A -85,B 0,C 180,E1 -16622.102,E2 -16622.102} C_VEL
LIN {X 0,Y 309.175,Z 306.877,A -85,B 0,C 180,E1 -16622.811,E2 -16622.811} C_VEL
LIN {X 0,Y 307.247,Z 366.919,A -85,B 0,C 180,E1 -16624.24,E2 -16624.24} C_VEL
LIN {X 0,Y 306.085,Z 380.695,A -85,B 0,C 180,E1 -16624.818,E2 -16624.818} C_VEL
LIN {X 0,Y 304.523,Z 393.595,A -85,B 0,C 180,E1 -16625.636,E2 -16625.636} C_VEL
LIN {X 0,Y 302.554,Z 406.122,A -85,B 0,C 180,E1 -16626.74,E2 -16626.74} C_VEL
LIN {X 0,Y 300.412,Z 417.31,A -85,B 0,C 180,E1 -16628.018,E2 -16628.018} C_VEL
LIN {X 0,Y 298.397,Z 427.407,A -85,B 0,C 180,E1 -16629.491,E2 -16629.491} C_VEL
LIN {X 0,Y 296.151,Z 437.345,A -85,B 0,C 180,E1 -16631.314,E2 -16631.314} C_VEL
LIN {X 0,Y 294.21,Z 446.124,A -85,B 0,C 180,E1 -16633.341,E2 -16633.341} C_VEL
LIN {X 0,Y 292.623,Z 453.18,A -85,B 0,C 180,E1 -16635.392,E2 -16635.392} C_VEL
LIN {X 0,Y 291.226,Z 458.845,A -85,B 0,C 180,E1 -16637.454,E2 -16637.454} C_VEL
LIN {X 0,Y 290.403,Z 463.336,A -85,B 0,C 180,E1 -16639.541,E2 -16639.541} C_VEL
LIN {X 0,Y 289.839,Z 466.769,A -85,B 0,C 180,E1 -16641.633,E2 -16641.633} C_VEL
LIN {X 0,Y 289.481,Z 469.813,A -85,B 0,C 180,E1 -16644.425,E2 -16644.425} C_VEL
LIN {X 0,Y 289.47,Z 470.747,A -85,B 0,C 180,E1 -16645.821,E2 -16645.821} C_VEL
LIN {X 0,Y 289.504,Z 471.268,A -85,B 0,C 180,E1 -16647.215,E2 -16647.215} C_VEL
LIN {X 0,Y 289.586,Z 471.084,A -85,B 0,C 180,E1 -16649.997,E2 -16649.997} C_VEL
LIN {X 0,Y 289.548,Z 470.404,A -85,B 0,C 180,E1 -16651.388,E2 -16651.388} C_VEL
LIN {X 0,Y 289.537,Z 469.309,A -85,B 0,C 180,E1 -16652.78,E2 -16652.78} C_VEL
LIN {X 0,Y 289.541,Z 467.757,A -85,B 0,C 180,E1 -16654.173,E2 -16654.173} C_VEL
LIN {X 0,Y 289.596,Z 464.749,A -85,B 0,C 180,E1 -16656.196,E2 -16656.196} C_VEL
LIN {X 0,Y 289.814,Z 460.405,A -85,B 0,C 180,E1 -16658.363,E2 -16658.363} C_VEL
LIN {X 0,Y 290.313,Z 453.958,A -85,B 0,C 180,E1 -16660.81,E2 -16660.81} C_VEL
LIN {X 0,Y 291.157,Z 446.929,A -85,B 0,C 180,E1 -16662.898,E2 -16662.898} C_VEL
LIN {X 0,Y 292.265,Z 438.093,A -85,B 0,C 180,E1 -16664.977,E2 -16664.977} C_VEL
LIN {X 0,Y 293.354,Z 429.023,A -85,B 0,C 180,E1 -16666.703,E2 -16666.703} C_VEL
LIN {X 0,Y 294.575,Z 419.044,A -85,B 0,C 180,E1 -16668.244,E2 -16668.244} C_VEL
LIN {X 0,Y 296.022,Z 408.011,A -85,B 0,C 180,E1 -16669.589,E2 -16669.589} C_VEL
LIN {X 0,Y 297.331,Z 395.602,A -85,B 0,C 180,E1 -16670.761,E2 -16670.761} C_VEL
LIN {X 0,Y 298.367,Z 383.855,A -85,B 0,C 180,E1 -16671.59,E2 -16671.59} C_VEL
LIN {X 0,Y 299.253,Z 371.41,A -85,B 0,C 180,E1 -16672.199,E2 -16672.199} C_VEL
LIN {X 0,Y 299.718,Z 355.901,A -85,B 0,C 180,E1 -16672.649,E2 -16672.649} C_VEL
LIN {X 0,Y 300.768,Z 302.844,A -85,B 0,C 180,E1 -16673.904,E2 -16673.904} C_VEL
LIN {X 0,Y 295.452,Z 261.733,A -85,B 0,C 180,E1 -16675.322,E2 -16675.322} C_VEL
LIN {X 0,Y 294.947,Z 258.146,A -85,B 0,C 180,E1 -16675.487,E2 -16675.487} C_VEL
LIN {X 0,Y 295.424,Z 252.985,A -85,B 0,C 180,E1 -16676.866,E2 -16676.866} C_VEL
LIN {X 0,Y 293.139,Z 241.161,A -85,B 0,C 180,E1 -16680.333,E2 -16680.333} C_VEL
LIN {X 0,Y 291.389,Z 233.192,A -85,B 0,C 180,E1 -16682.813,E2 -16682.813} C_VEL
LIN {X 0,Y 291.362,Z 233.192,A -85,B 0,C 180,E1 -16687.25,E2 -16687.25} C_VEL
LIN {X 0,Y 291.313,Z 233.196,A -85,B 0,C 180,E1 -16690.638,E2 -16690.638} C_VEL
LIN {X 0,Y 291.291,Z 233.199,A -85,B 0,C 180,E1 -16694.393,E2 -16694.393} C_VEL
LIN {X 0,Y 291.354,Z 233.192,A -85,B 0,C 180,E1 -16698.388,E2 -16698.388} C_VEL
LIN {X 0,Y 291.348,Z 233.192,A -85,B 0,C 180,E1 -16701.158,E2 -16701.158} C_VEL
LIN {X 0,Y 291.337,Z 233.193,A -85,B 0,C 180,E1 -16704.623,E2 -16704.623} C_VEL
LIN {X 0,Y 291.338,Z 233.195,A -85,B 0,C 180,E1 -16707.947,E2 -16707.947} C_VEL
LIN {X 0,Y 291.347,Z 233.193,A -85,B 0,C 180,E1 -16711.155,E2 -16711.155} C_VEL
LIN {X 0,Y 291.387,Z 233.186,A -85,B 0,C 180,E1 -16714.269,E2 -16714.269} C_VEL
LIN {X 0,Y 291.402,Z 233.188,A -85,B 0,C 180,E1 -16717.301,E2 -16717.301} C_VEL
LIN {X 0,Y 291.467,Z 233.176,A -85,B 0,C 180,E1 -16720.271,E2 -16720.271} C_VEL
LIN {X 0,Y 291.477,Z 233.175,A -85,B 0,C 180,E1 -16724.65,E2 -16724.65} C_VEL
LIN {X 0,Y 291.494,Z 233.174,A -85,B 0,C 180,E1 -16728.879,E2 -16728.879} C_VEL
LIN {X 0,Y 291.659,Z 233.151,A -85,B 0,C 180,E1 -16731.687,E2 -16731.687} C_VEL
LIN {X 0,Y 291.588,Z 233.16,A -85,B 0,C 180,E1 -16734.468,E2 -16734.468} C_VEL
LIN {X 0,Y 291.844,Z 233.129,A -85,B 0,C 180,E1 -16738.62,E2 -16738.62} C_VEL
LIN {X 0,Y 291.843,Z 233.118,A -85,B 0,C 180,E1 -16741.38,E2 -16741.38} C_VEL
LIN {X 0,Y 291.686,Z 233.152,A -85,B 0,C 180,E1 -16746.92,E2 -16746.92} C_VEL
LIN {X 0,Y 291.53,Z 233.167,A -85,B 0,C 180,E1 -16749.715,E2 -16749.715} C_VEL
LIN {X 0,Y 291.473,Z 233.165,A -85,B 0,C 180,E1 -16753.953,E2 -16753.953} C_VEL
LIN {X 0,Y 291.39,Z 233.184,A -85,B 0,C 180,E1 -16756.824,E2 -16756.824} C_VEL
LIN {X 0,Y 291.354,Z 233.19,A -85,B 0,C 180,E1 -16759.845,E2 -16759.845} C_VEL
LIN {X 0,Y 291.345,Z 233.191,A -85,B 0,C 180,E1 -16764.21,E2 -16764.21} C_VEL
LIN {X 0,Y 291.382,Z 233.187,A -85,B 0,C 180,E1 -16767.276,E2 -16767.276} C_VEL
LIN {X 0,Y 291.303,Z 233.199,A -85,B 0,C 180,E1 -16770.441,E2 -16770.441} C_VEL
LIN {X 0,Y 291.313,Z 233.195,A -85,B 0,C 180,E1 -16773.703,E2 -16773.703} C_VEL
LIN {X 0,Y 291.368,Z 233.188,A -85,B 0,C 180,E1 -16777.264,E2 -16777.264} C_VEL
LIN {X 0,Y 291.374,Z 233.19,A -85,B 0,C 180,E1 -16780.636,E2 -16780.636} C_VEL
LIN {X 0,Y 291.31,Z 233.193,A -85,B 0,C 180,E1 -16784.398,E2 -16784.398} C_VEL
LIN {X 0,Y 291.306,Z 233.199,A -85,B 0,C 180,E1 -16788.409,E2 -16788.409} C_VEL
LIN {X 0,Y 291.329,Z 233.191,A -85,B 0,C 180,E1 -16791.162,E2 -16791.162} C_VEL
LIN {X 0,Y 291.345,Z 233.192,A -85,B 0,C 180,E1 -16794.631,E2 -16794.631} C_VEL
LIN {X 0,Y 291.357,Z 233.193,A -85,B 0,C 180,E1 -16797.955,E2 -16797.955} C_VEL
LIN {X 0,Y 291.366,Z 233.189,A -85,B 0,C 180,E1 -16801.163,E2 -16801.163} C_VEL
LIN {X 0,Y 291.406,Z 233.185,A -85,B 0,C 180,E1 -16804.277,E2 -16804.277} C_VEL
LIN {X 0,Y 291.365,Z 233.189,A -85,B 0,C 180,E1 -16807.303,E2 -16807.303} C_VEL
LIN {X 0,Y 291.401,Z 233.186,A -85,B 0,C 180,E1 -16810.271,E2 -16810.271} C_VEL
LIN {X 0,Y 291.58,Z 233.239,A -85,B 0,C 180,E1 -16815.21,E2 -16815.21} C_VEL
LIN {X 0,Y 291.671,Z 233.77,A -85,B 0,C 180,E1 -16815.382,E2 -16815.382} C_VEL
LIN {X 0,Y 300.544,Z 258.544,A -85,B 0,C 180,E1 -16816.691,E2 -16816.691} C_VEL
LIN {X 0,Y 301.619,Z 263.247,A -85,B 0,C 180,E1 -16816.886,E2 -16816.886} C_VEL
LIN {X 0,Y 299.72,Z 340.667,A -85,B 0,C 180,E1 -16818.721,E2 -16818.721} C_VEL
LIN {X 0,Y 299.003,Z 353.997,A -85,B 0,C 180,E1 -16819.294,E2 -16819.294} C_VEL
LIN {X 0,Y 298.249,Z 366.109,A -85,B 0,C 180,E1 -16820.081,E2 -16820.081} C_VEL
LIN {X 0,Y 297.497,Z 376.634,A -85,B 0,C 180,E1 -16820.999,E2 -16820.999} C_VEL
LIN {X 0,Y 296.293,Z 387.321,A -85,B 0,C 180,E1 -16822.164,E2 -16822.164} C_VEL
LIN {X 0,Y 295.105,Z 397.141,A -85,B 0,C 180,E1 -16823.508,E2 -16823.508} C_VEL
LIN {X 0,Y 293.788,Z 407.076,A -85,B 0,C 180,E1 -16825.2,E2 -16825.2} C_VEL
LIN {X 0,Y 292.572,Z 416.688,A -85,B 0,C 180,E1 -16827.249,E2 -16827.249} C_VEL
LIN {X 0,Y 291.463,Z 424.372,A -85,B 0,C 180,E1 -16829.312,E2 -16829.312} C_VEL
LIN {X 0,Y 290.788,Z 430.521,A -85,B 0,C 180,E1 -16831.387,E2 -16831.387} C_VEL
LIN {X 0,Y 290.205,Z 435.423,A -85,B 0,C 180,E1 -16833.473,E2 -16833.473} C_VEL
LIN {X 0,Y 289.917,Z 439.202,A -85,B 0,C 180,E1 -16835.567,E2 -16835.567} C_VEL
LIN {X 0,Y 289.723,Z 441.164,A -85,B 0,C 180,E1 -16836.968,E2 -16836.968} C_VEL
LIN {X 0,Y 289.535,Z 442.712,A -85,B 0,C 180,E1 -16838.376,E2 -16838.376} C_VEL
LIN {X 0,Y 289.441,Z 443.801,A -85,B 0,C 180,E1 -16839.788,E2 -16839.788} C_VEL
LIN {X 0,Y 289.519,Z 444.794,A -85,B 0,C 180,E1 -16842.621,E2 -16842.621} C_VEL
LIN {X 0,Y 289.689,Z 444.692,A -85,B 0,C 180,E1 -16844.042,E2 -16844.042} C_VEL
LIN {X 0,Y 289.846,Z 444.149,A -85,B 0,C 180,E1 -16845.47,E2 -16845.47} C_VEL
LIN {X 0,Y 290.128,Z 443.205,A -85,B 0,C 180,E1 -16846.9,E2 -16846.9} C_VEL
LIN {X 0,Y 290.571,Z 441.854,A -85,B 0,C 180,E1 -16848.327,E2 -16848.327} C_VEL
LIN {X 0,Y 291.369,Z 438.958,A -85,B 0,C 180,E1 -16850.473,E2 -16850.473} C_VEL
LIN {X 0,Y 292.396,Z 434.977,A -85,B 0,C 180,E1 -16852.618,E2 -16852.618} C_VEL
LIN {X 0,Y 293.822,Z 429.482,A -85,B 0,C 180,E1 -16854.855,E2 -16854.855} C_VEL
LIN {X 0,Y 295.435,Z 423.15,A -85,B 0,C 180,E1 -16856.871,E2 -16856.871} C_VEL
LIN {X 0,Y 297.404,Z 415.153,A -85,B 0,C 180,E1 -16858.896,E2 -16858.896} C_VEL
LIN {X 0,Y 299.353,Z 406.276,A -85,B 0,C 180,E1 -16860.706,E2 -16860.706} C_VEL
LIN {X 0,Y 301.277,Z 396.806,A -85,B 0,C 180,E1 -16862.249,E2 -16862.249} C_VEL
LIN {X 0,Y 303.171,Z 386.756,A -85,B 0,C 180,E1 -16863.558,E2 -16863.558} C_VEL
LIN {X 0,Y 304.847,Z 374.951,A -85,B 0,C 180,E1 -16864.791,E2 -16864.791} C_VEL
LIN {X 0,Y 306.093,Z 364.428,A -85,B 0,C 180,E1 -16865.634,E2 -16865.634} C_VEL
LIN {X 0,Y 307.314,Z 351.62,A -85,B 0,C 180,E1 -16866.381,E2 -16866.381} C_VEL
LIN {X 0,Y 308.032,Z 339.037,A -85,B 0,C 180,E1 -16866.856,E2 -16866.856} C_VEL
LIN {X 0,Y 310.24,Z 272.243,A -85,B 0,C 180,E1 -16868.41,E2 -16868.41} C_VEL
LIN {X 0,Y 303.76,Z 257.686,A -85,B 0,C 180,E1 -16869.574,E2 -16869.574} C_VEL
LIN {X 0,Y 295.895,Z 242.419,A -85,B 0,C 180,E1 -16871.011,E2 -16871.011} C_VEL
LIN {X 0,Y 291.787,Z 234.817,A -85,B 0,C 180,E1 -16871.821,E2 -16871.821} C_VEL
LIN {X 0,Y 291.405,Z 233.19,A -85,B 0,C 180,E1 -16872.475,E2 -16872.475} C_VEL
LIN {X 0,Y 291.367,Z 233.195,A -85,B 0,C 180,E1 -16876.352,E2 -16876.352} C_VEL
LIN {X 0,Y 291.395,Z 233.186,A -85,B 0,C 180,E1 -16880.512,E2 -16880.512} C_VEL
LIN {X 0,Y 291.345,Z 233.19,A -85,B 0,C 180,E1 -16884.327,E2 -16884.327} C_VEL
LIN {X 0,Y 290.715,Z 233.278,A -85,B 0,C 180,E1 -16885.48,E2 -16885.48} C_VEL
LIN {X 0,Y 287.929,Z 233.635,A -85,B 0,C 180,E1 -16887.359,E2 -16887.359} C_VEL
LIN {X 0,Y 285.523,Z 233.932,A -85,B 0,C 180,E1 -16888.883,E2 -16888.883} C_VEL
LIN {X 0,Y 284.449,Z 234.057,A -85,B 0,C 180,E1 -16890.063,E2 -16890.063} C_VEL
LIN {X 0,Y 284.34,Z 234.066,A -85,B 0,C 180,E1 -16890.464,E2 -16890.464} C_VEL
LIN {X 0,Y 284.365,Z 234.058,A -85,B 0,C 180,E1 -16893.585,E2 -16893.585} C_VEL
LIN {X 0,Y 284.319,Z 234.06,A -85,B 0,C 180,E1 -16896.703,E2 -16896.703} C_VEL
LIN {X 0,Y 284.364,Z 234.054,A -85,B 0,C 180,E1 -16899.904,E2 -16899.904} C_VEL
LIN {X 0,Y 284.434,Z 234.044,A -85,B 0,C 180,E1 -16904.491,E2 -16904.491} C_VEL
LIN {X 0,Y 284.45,Z 234.045,A -85,B 0,C 180,E1 -16908.6,E2 -16908.6} C_VEL
LIN {X 0,Y 284.616,Z 234.033,A -85,B 0,C 180,E1 -16911.48,E2 -16911.48} C_VEL
LIN {X 0,Y 284.575,Z 234.03,A -85,B 0,C 180,E1 -16914.331,E2 -16914.331} C_VEL
LIN {X 0,Y 284.834,Z 233.993,A -85,B 0,C 180,E1 -16918.586,E2 -16918.586} C_VEL
LIN {X 0,Y 284.834,Z 234.002,A -85,B 0,C 180,E1 -16921.414,E2 -16921.414} C_VEL
LIN {X 0,Y 284.621,Z 234.021,A -85,B 0,C 180,E1 -16927.092,E2 -16927.092} C_VEL
LIN {X 0,Y 284.495,Z 234.045,A -85,B 0,C 180,E1 -16929.958,E2 -16929.958} C_VEL
LIN {X 0,Y 284.446,Z 234.051,A -85,B 0,C 180,E1 -16934.304,E2 -16934.304} C_VEL
LIN {X 0,Y 284.314,Z 234.068,A -85,B 0,C 180,E1 -16938.744,E2 -16938.744} C_VEL
LIN {X 0,Y 284.296,Z 234.072,A -85,B 0,C 180,E1 -16943.299,E2 -16943.299} C_VEL
LIN {X 0,Y 284.274,Z 234.074,A -85,B 0,C 180,E1 -16947.13,E2 -16947.13} C_VEL
LIN {X 0,Y 284.26,Z 234.067,A -85,B 0,C 180,E1 -16950.083,E2 -16950.083} C_VEL
LIN {X 0,Y 284.274,Z 234.067,A -85,B 0,C 180,E1 -16952.949,E2 -16952.949} C_VEL
LIN {X 0,Y 284.31,Z 234.062,A -85,B 0,C 180,E1 -16956.389,E2 -16956.389} C_VEL
LIN {X 0,Y 284.299,Z 234.055,A -85,B 0,C 180,E1 -16959.996,E2 -16959.996} C_VEL
LIN {X 0,Y 284.241,Z 234.081,A -85,B 0,C 180,E1 -16964.191,E2 -16964.191} C_VEL
LIN {X 0,Y 284.234,Z 234.067,A -85,B 0,C 180,E1 -16968.119,E2 -16968.119} C_VEL
LIN {X 0,Y 284.33,Z 234.234,A -85,B 0,C 180,E1 -16970.815,E2 -16970.815} C_VEL
LIN {X 0,Y 286.893,Z 243.488,A -85,B 0,C 180,E1 -16974.37,E2 -16974.37} C_VEL
LIN {X 0,Y 289.093,Z 252.771,A -85,B 0,C 180,E1 -16977.668,E2 -16977.668} C_VEL
LIN {X 0,Y 290.021,Z 256.93,A -85,B 0,C 180,E1 -16979.035,E2 -16979.035} C_VEL
LIN {X 0,Y 296.637,Z 271.558,A -85,B 0,C 180,E1 -16980.341,E2 -16980.341} C_VEL
LIN {X 0,Y 300.52,Z 291.358,A -85,B 0,C 180,E1 -16981.384,E2 -16981.384} C_VEL
LIN {X 0,Y 303.062,Z 308.31,A -85,B 0,C 180,E1 -16982.156,E2 -16982.156} C_VEL
LIN {X 0,Y 301.089,Z 366.925,A -85,B 0,C 180,E1 -16983.581,E2 -16983.581} C_VEL
LIN {X 0,Y 299.884,Z 380.567,A -85,B 0,C 180,E1 -16984.166,E2 -16984.166} C_VEL
LIN {X 0,Y 298.265,Z 393.398,A -85,B 0,C 180,E1 -16984.997,E2 -16984.997} C_VEL
LIN {X 0,Y 296.333,Z 405.113,A -85,B 0,C 180,E1 -16986.037,E2 -16986.037} C_VEL
LIN {X 0,Y 294.146,Z 416.422,A -85,B 0,C 180,E1 -16987.339,E2 -16987.339} C_VEL
LIN {X 0,Y 291.97,Z 426.643,A -85,B 0,C 180,E1 -16988.834,E2 -16988.834} C_VEL
LIN {X 0,Y 289.851,Z 435.849,A -85,B 0,C 180,E1 -16990.524,E2 -16990.524} C_VEL
LIN {X 0,Y 287.954,Z 443.836,A -85,B 0,C 180,E1 -16992.336,E2 -16992.336} C_VEL
LIN {X 0,Y 286.286,Z 450.959,A -85,B 0,C 180,E1 -16994.332,E2 -16994.332} C_VEL
LIN {X 0,Y 284.73,Z 457.006,A -85,B 0,C 180,E1 -16996.437,E2 -16996.437} C_VEL
LIN {X 0,Y 283.655,Z 461.819,A -85,B 0,C 180,E1 -16998.566,E2 -16998.566} C_VEL
LIN {X 0,Y 282.946,Z 465.537,A -85,B 0,C 180,E1 -17000.707,E2 -17000.707} C_VEL
LIN {X 0,Y 282.509,Z 468.259,A -85,B 0,C 180,E1 -17002.853,E2 -17002.853} C_VEL
LIN {X 0,Y 282.41,Z 469.754,A -85,B 0,C 180,E1 -17004.524,E2 -17004.524} C_VEL
LIN {X 0,Y 282.429,Z 470.952,A -85,B 0,C 180,E1 -17007.145,E2 -17007.145} C_VEL
LIN {X 0,Y 282.499,Z 470.725,A -85,B 0,C 180,E1 -17009.997,E2 -17009.997} C_VEL
LIN {X 0,Y 282.464,Z 470.023,A -85,B 0,C 180,E1 -17011.423,E2 -17011.423} C_VEL
LIN {X 0,Y 282.463,Z 468.884,A -85,B 0,C 180,E1 -17012.849,E2 -17012.849} C_VEL
LIN {X 0,Y 282.441,Z 467.307,A -85,B 0,C 180,E1 -17014.278,E2 -17014.278} C_VEL
LIN {X 0,Y 282.528,Z 464.126,A -85,B 0,C 180,E1 -17016.424,E2 -17016.424} C_VEL
LIN {X 0,Y 282.751,Z 459.855,A -85,B 0,C 180,E1 -17018.573,E2 -17018.573} C_VEL
LIN {X 0,Y 283.264,Z 453.351,A -85,B 0,C 180,E1 -17021.082,E2 -17021.082} C_VEL
LIN {X 0,Y 284.202,Z 446.236,A -85,B 0,C 180,E1 -17023.219,E2 -17023.219} C_VEL
LIN {X 0,Y 285.381,Z 437.315,A -85,B 0,C 180,E1 -17025.347,E2 -17025.347} C_VEL
LIN {X 0,Y 286.33,Z 429.327,A -85,B 0,C 180,E1 -17026.906,E2 -17026.906} C_VEL
LIN {X 0,Y 287.629,Z 419.244,A -85,B 0,C 180,E1 -17028.516,E2 -17028.516} C_VEL
LIN {X 0,Y 289.105,Z 408.386,A -85,B 0,C 180,E1 -17029.892,E2 -17029.892} C_VEL
LIN {X 0,Y 290.463,Z 396.158,A -85,B 0,C 180,E1 -17031.09,E2 -17031.09} C_VEL
LIN {X 0,Y 291.636,Z 383.365,A -85,B 0,C 180,E1 -17032.021,E2 -17032.021} C_VEL
LIN {X 0,Y 292.533,Z 370.827,A -85,B 0,C 180,E1 -17032.642,E2 -17032.642} C_VEL
LIN {X 0,Y 293.006,Z 355.302,A -85,B 0,C 180,E1 -17033.099,E2 -17033.099} C_VEL
LIN {X 0,Y 294.092,Z 303.679,A -85,B 0,C 180,E1 -17034.345,E2 -17034.345} C_VEL
LIN {X 0,Y 288.706,Z 261.891,A -85,B 0,C 180,E1 -17035.832,E2 -17035.832} C_VEL
LIN {X 0,Y 288.137,Z 257.949,A -85,B 0,C 180,E1 -17035.983,E2 -17035.983} C_VEL
LIN {X 0,Y 288.485,Z 255.014,A -85,B 0,C 180,E1 -17036.782,E2 -17036.782} C_VEL
LIN {X 0,Y 286.719,Z 245.12,A -85,B 0,C 180,E1 -17039.727,E2 -17039.727} C_VEL
LIN {X 0,Y 284.314,Z 234.074,A -85,B 0,C 180,E1 -17043.254,E2 -17043.254} C_VEL
LIN {X 0,Y 284.316,Z 234.071,A -85,B 0,C 180,E1 -17046.381,E2 -17046.381} C_VEL
LIN {X 0,Y 284.286,Z 234.076,A -85,B 0,C 180,E1 -17049.99,E2 -17049.99} C_VEL
LIN {X 0,Y 284.243,Z 234.078,A -85,B 0,C 180,E1 -17054.19,E2 -17054.19} C_VEL
LIN {X 0,Y 284.303,Z 234.072,A -85,B 0,C 180,E1 -17058.13,E2 -17058.13} C_VEL
LIN {X 0,Y 284.299,Z 234.073,A -85,B 0,C 180,E1 -17061.829,E2 -17061.829} C_VEL
LIN {X 0,Y 284.28,Z 234.075,A -85,B 0,C 180,E1 -17065.347,E2 -17065.347} C_VEL
LIN {X 0,Y 284.262,Z 234.074,A -85,B 0,C 180,E1 -17068.722,E2 -17068.722} C_VEL
LIN {X 0,Y 284.363,Z 234.062,A -85,B 0,C 180,E1 -17072.823,E2 -17072.823} C_VEL
LIN {X 0,Y 284.36,Z 234.061,A -85,B 0,C 180,E1 -17076.706,E2 -17076.706} C_VEL
LIN {X 0,Y 284.395,Z 234.058,A -85,B 0,C 180,E1 -17079.871,E2 -17079.871} C_VEL
LIN {X 0,Y 284.416,Z 234.055,A -85,B 0,C 180,E1 -17084.484,E2 -17084.484} C_VEL
LIN {X 0,Y 284.446,Z 234.05,A -85,B 0,C 180,E1 -17088.6,E2 -17088.6} C_VEL
LIN {X 0,Y 284.609,Z 234.031,A -85,B 0,C 180,E1 -17091.48,E2 -17091.48} C_VEL
LIN {X 0,Y 284.559,Z 234.035,A -85,B 0,C 180,E1 -17094.331,E2 -17094.331} C_VEL
LIN {X 0,Y 284.811,Z 234.004,A -85,B 0,C 180,E1 -17098.586,E2 -17098.586} C_VEL
LIN {X 0,Y 284.809,Z 233.993,A -85,B 0,C 180,E1 -17101.414,E2 -17101.414} C_VEL
LIN {X 0,Y 284.637,Z 234.03,A -85,B 0,C 180,E1 -17107.092,E2 -17107.092} C_VEL
LIN {X 0,Y 284.476,Z 234.046,A -85,B 0,C 180,E1 -17109.959,E2 -17109.959} C_VEL
LIN {X 0,Y 284.422,Z 234.043,A -85,B 0,C 180,E1 -17114.306,E2 -17114.306} C_VEL
LIN {X 0,Y 284.294,Z 234.072,A -85,B 0,C 180,E1 -17118.746,E2 -17118.746} C_VEL
LIN {X 0,Y 284.295,Z 234.068,A -85,B 0,C 180,E1 -17123.299,E2 -17123.299} C_VEL
LIN {X 0,Y 284.359,Z 234.062,A -85,B 0,C 180,E1 -17127.175,E2 -17127.175} C_VEL
LIN {X 0,Y 284.262,Z 234.074,A -85,B 0,C 180,E1 -17131.279,E2 -17131.279} C_VEL
LIN {X 0,Y 284.316,Z 234.066,A -85,B 0,C 180,E1 -17135.353,E2 -17135.353} C_VEL
LIN {X 0,Y 284.302,Z 234.072,A -85,B 0,C 180,E1 -17138.171,E2 -17138.171} C_VEL
LIN {X 0,Y 284.303,Z 234.071,A -85,B 0,C 180,E1 -17142.142,E2 -17142.142} C_VEL
LIN {X 0,Y 284.247,Z 234.071,A -85,B 0,C 180,E1 -17146.197,E2 -17146.197} C_VEL
LIN {X 0,Y 284.288,Z 234.073,A -85,B 0,C 180,E1 -17150.029,E2 -17150.029} C_VEL
LIN {X 0,Y 284.313,Z 234.063,A -85,B 0,C 180,E1 -17153.619,E2 -17153.619} C_VEL
LIN {X 0,Y 284.293,Z 234.069,A -85,B 0,C 180,E1 -17157.195,E2 -17157.195} C_VEL
LIN {X 0,Y 284.343,Z 234.066,A -85,B 0,C 180,E1 -17160.381,E2 -17160.381} C_VEL
LIN {X 0,Y 284.368,Z 234.063,A -85,B 0,C 180,E1 -17163.591,E2 -17163.591} C_VEL
LIN {X 0,Y 284.325,Z 234.065,A -85,B 0,C 180,E1 -17166.709,E2 -17166.709} C_VEL
LIN {X 0,Y 284.371,Z 234.063,A -85,B 0,C 180,E1 -17169.909,E2 -17169.909} C_VEL
LIN {X 0,Y 284.481,Z 234.05,A -85,B 0,C 180,E1 -17174.776,E2 -17174.776} C_VEL
LIN {X 0,Y 285.485,Z 236.903,A -85,B 0,C 180,E1 -17174.968,E2 -17174.968} C_VEL
LIN {X 0,Y 292.624,Z 256.157,A -85,B 0,C 180,E1 -17176.042,E2 -17176.042} C_VEL
LIN {X 0,Y 294.864,Z 263.477,A -85,B 0,C 180,E1 -17176.401,E2 -17176.401} C_VEL
LIN {X 0,Y 294.407,Z 285.533,A -85,B 0,C 180,E1 -17176.934,E2 -17176.934} C_VEL
LIN {X 0,Y 293.006,Z 340.93,A -85,B 0,C 180,E1 -17178.284,E2 -17178.284} C_VEL
LIN {X 0,Y 292.268,Z 354.282,A -85,B 0,C 180,E1 -17178.869,E2 -17178.869} C_VEL
LIN {X 0,Y 291.485,Z 366.404,A -85,B 0,C 180,E1 -17179.673,E2 -17179.673} C_VEL
LIN {X 0,Y 290.567,Z 378.635,A -85,B 0,C 180,E1 -17180.783,E2 -17180.783} C_VEL
LIN {X 0,Y 289.105,Z 390.243,A -85,B 0,C 180,E1 -17182.144,E2 -17182.144} C_VEL
LIN {X 0,Y 287.797,Z 400.649,A -85,B 0,C 180,E1 -17183.694,E2 -17183.694} C_VEL
LIN {X 0,Y 286.496,Z 410.035,A -85,B 0,C 180,E1 -17185.43,E2 -17185.43} C_VEL
LIN {X 0,Y 285.319,Z 419.061,A -85,B 0,C 180,E1 -17187.532,E2 -17187.532} C_VEL
LIN {X 0,Y 284.237,Z 426.363,A -85,B 0,C 180,E1 -17189.649,E2 -17189.649} C_VEL
LIN {X 0,Y 283.679,Z 431.298,A -85,B 0,C 180,E1 -17191.422,E2 -17191.422} C_VEL
LIN {X 0,Y 283.093,Z 436.106,A -85,B 0,C 180,E1 -17193.561,E2 -17193.561} C_VEL
LIN {X 0,Y 282.808,Z 439.797,A -85,B 0,C 180,E1 -17195.707,E2 -17195.707} C_VEL
LIN {X 0,Y 282.596,Z 441.718,A -85,B 0,C 180,E1 -17197.145,E2 -17197.145} C_VEL
LIN {X 0,Y 282.442,Z 443.189,A -85,B 0,C 180,E1 -17198.588,E2 -17198.588} C_VEL
LIN {X 0,Y 282.366,Z 444.883,A -85,B 0,C 180,E1 -17201.487,E2 -17201.487} C_VEL
LIN {X 0,Y 282.611,Z 445.045,A -85,B 0,C 180,E1 -17204.102,E2 -17204.102} C_VEL
LIN {X 0,Y 282.82,Z 444.381,A -85,B 0,C 180,E1 -17205.865,E2 -17205.865} C_VEL
LIN {X 0,Y 283.15,Z 443.396,A -85,B 0,C 180,E1 -17207.329,E2 -17207.329} C_VEL
LIN {X 0,Y 284.06,Z 440.589,A -85,B 0,C 180,E1 -17209.919,E2 -17209.919} C_VEL
LIN {X 0,Y 285.215,Z 436.393,A -85,B 0,C 180,E1 -17212.454,E2 -17212.454} C_VEL
LIN {X 0,Y 286.773,Z 430.756,A -85,B 0,C 180,E1 -17214.937,E2 -17214.937} C_VEL
LIN {X 0,Y 288.586,Z 424.114,A -85,B 0,C 180,E1 -17217.169,E2 -17217.169} C_VEL
LIN {X 0,Y 290.779,Z 415.595,A -85,B 0,C 180,E1 -17219.393,E2 -17219.393} C_VEL
LIN {X 0,Y 292.64,Z 407.528,A -85,B 0,C 180,E1 -17221.087,E2 -17221.087} C_VEL
LIN {X 0,Y 294.613,Z 398.297,A -85,B 0,C 180,E1 -17222.664,E2 -17222.664} C_VEL
LIN {X 0,Y 296.736,Z 387.73,A -85,B 0,C 180,E1 -17224.093,E2 -17224.093} C_VEL
LIN {X 0,Y 298.592,Z 375.3,A -85,B 0,C 180,E1 -17225.422,E2 -17225.422} C_VEL
LIN {X 0,Y 299.892,Z 364.782,A -85,B 0,C 180,E1 -17226.279,E2 -17226.279} C_VEL
LIN {X 0,Y 301.152,Z 351.991,A -85,B 0,C 180,E1 -17227.04,E2 -17227.04} C_VEL
LIN {X 0,Y 301.873,Z 340.242,A -85,B 0,C 180,E1 -17227.5,E2 -17227.5} C_VEL
LIN {X 0,Y 304.144,Z 274.12,A -85,B 0,C 180,E1 -17229.073,E2 -17229.073} C_VEL
LIN {X 0,Y 297.511,Z 259.452,A -85,B 0,C 180,E1 -17230.308,E2 -17230.308} C_VEL
LIN {X 0,Y 290.368,Z 245.738,A -85,B 0,C 180,E1 -17231.665,E2 -17231.665} C_VEL
LIN {X 0,Y 284.579,Z 235.167,A -85,B 0,C 180,E1 -17232.866,E2 -17232.866} C_VEL
LIN {X 0,Y 284.347,Z 234.057,A -85,B 0,C 180,E1 -17233.356,E2 -17233.356} C_VEL
LIN {X 0,Y 284.336,Z 234.066,A -85,B 0,C 180,E1 -17237.859,E2 -17237.859} C_VEL
LIN {X 0,Y 284.32,Z 234.067,A -85,B 0,C 180,E1 -17241.832,E2 -17241.832} C_VEL
LIN {X 0,Y 284.3,Z 234.066,A -85,B 0,C 180,E1 -17245.349,E2 -17245.349} C_VEL
LIN {X 0,Y 284.285,Z 234.066,A -85,B 0,C 180,E1 -17248.724,E2 -17248.724} C_VEL
LIN {X 0,Y 284.34,Z 234.066,A -85,B 0,C 180,E1 -17250.464,E2 -17250.464} C_VEL
LIN {X 0,Y 283.619,Z 234.153,A -85,B 0,C 180,E1 -17251.646,E2 -17251.646} C_VEL
LIN {X 0,Y 280.764,Z 234.507,A -85,B 0,C 180,E1 -17253.574,E2 -17253.574} C_VEL
LIN {X 0,Y 278.37,Z 234.809,A -85,B 0,C 180,E1 -17255.139,E2 -17255.139} C_VEL
LIN {X 0,Y 277.335,Z 234.93,A -85,B 0,C 180,E1 -17256.351,E2 -17256.351} C_VEL
LIN {X 0,Y 277.244,Z 234.94,A -85,B 0,C 180,E1 -17256.762,E2 -17256.762} C_VEL
LIN {X 0,Y 277.313,Z 234.931,A -85,B 0,C 180,E1 -17260.764,E2 -17260.764} C_VEL
LIN {X 0,Y 277.394,Z 234.922,A -85,B 0,C 180,E1 -17265.323,E2 -17265.323} C_VEL
LIN {X 0,Y 277.44,Z 234.919,A -85,B 0,C 180,E1 -17269.786,E2 -17269.786} C_VEL
LIN {X 0,Y 277.619,Z 234.898,A -85,B 0,C 180,E1 -17272.728,E2 -17272.728} C_VEL
LIN {X 0,Y 277.8,Z 234.869,A -85,B 0,C 180,E1 -17278.55,E2 -17278.55} C_VEL
LIN {X 0,Y 277.8,Z 234.878,A -85,B 0,C 180,E1 -17281.45,E2 -17281.45} C_VEL
LIN {X 0,Y 277.577,Z 234.897,A -85,B 0,C 180,E1 -17287.273,E2 -17287.273} C_VEL
LIN {X 0,Y 277.437,Z 234.925,A -85,B 0,C 180,E1 -17290.214,E2 -17290.214} C_VEL
LIN {X 0,Y 277.393,Z 234.932,A -85,B 0,C 180,E1 -17294.676,E2 -17294.676} C_VEL
LIN {X 0,Y 277.269,Z 234.947,A -85,B 0,C 180,E1 -17299.239,E2 -17299.239} C_VEL
LIN {X 0,Y 277.246,Z 234.95,A -85,B 0,C 180,E1 -17303.928,E2 -17303.928} C_VEL
LIN {X 0,Y 277.223,Z 234.953,A -85,B 0,C 180,E1 -17307.469,E2 -17307.469} C_VEL
LIN {X 0,Y 277.219,Z 234.946,A -85,B 0,C 180,E1 -17310.467,E2 -17310.467} C_VEL
LIN {X 0,Y 277.229,Z 234.943,A -85,B 0,C 180,E1 -17313.898,E2 -17313.898} C_VEL
LIN {X 0,Y 277.244,Z 234.927,A -85,B 0,C 180,E1 -17317.473,E2 -17317.473} C_VEL
LIN {X 0,Y 277.194,Z 234.957,A -85,B 0,C 180,E1 -17321.239,E2 -17321.239} C_VEL
LIN {X 0,Y 277.19,Z 234.953,A -85,B 0,C 180,E1 -17325.229,E2 -17325.229} C_VEL
LIN {X 0,Y 277.215,Z 234.951,A -85,B 0,C 180,E1 -17329.719,E2 -17329.719} C_VEL
LIN {X 0,Y 277.323,Z 235.411,A -85,B 0,C 180,E1 -17330.012,E2 -17330.012} C_VEL
LIN {X 0,Y 279.784,Z 244.095,A -85,B 0,C 180,E1 -17333.497,E2 -17333.497} C_VEL
LIN {X 0,Y 281.944,Z 252.857,A -85,B 0,C 180,E1 -17336.744,E2 -17336.744} C_VEL
LIN {X 0,Y 282.746,Z 256.498,A -85,B 0,C 180,E1 -17337.986,E2 -17337.986} C_VEL
LIN {X 0,Y 290.826,Z 274,A -85,B 0,C 180,E1 -17339.65,E2 -17339.65} C_VEL
LIN {X 0,Y 293.313,Z 285.998,A -85,B 0,C 180,E1 -17340.329,E2 -17340.329} C_VEL
LIN {X 0,Y 296.742,Z 306.442,A -85,B 0,C 180,E1 -17341.347,E2 -17341.347} C_VEL
LIN {X 0,Y 296.985,Z 310.623,A -85,B 0,C 180,E1 -17341.495,E2 -17341.495} C_VEL
LIN {X 0,Y 294.989,Z 366.613,A -85,B 0,C 180,E1 -17342.88,E2 -17342.88} C_VEL
LIN {X 0,Y 293.718,Z 380.481,A -85,B 0,C 180,E1 -17343.487,E2 -17343.487} C_VEL
LIN {X 0,Y 292.033,Z 393.223,A -85,B 0,C 180,E1 -17344.33,E2 -17344.33} C_VEL
LIN {X 0,Y 289.903,Z 405.687,A -85,B 0,C 180,E1 -17345.471,E2 -17345.471} C_VEL
LIN {X 0,Y 287.628,Z 416.828,A -85,B 0,C 180,E1 -17346.796,E2 -17346.796} C_VEL
LIN {X 0,Y 285.362,Z 426.879,A -85,B 0,C 180,E1 -17348.319,E2 -17348.319} C_VEL
LIN {X 0,Y 283.159,Z 435.98,A -85,B 0,C 180,E1 -17350.045,E2 -17350.045} C_VEL
LIN {X 0,Y 281.063,Z 444.394,A -85,B 0,C 180,E1 -17352.028,E2 -17352.028} C_VEL
LIN {X 0,Y 279.178,Z 452.064,A -85,B 0,C 180,E1 -17354.298,E2 -17354.298} C_VEL
LIN {X 0,Y 277.334,Z 458.642,A -85,B 0,C 180,E1 -17356.815,E2 -17356.815} C_VEL
LIN {X 0,Y 276.371,Z 463.026,A -85,B 0,C 180,E1 -17359.003,E2 -17359.003} C_VEL
LIN {X 0,Y 275.728,Z 466.359,A -85,B 0,C 180,E1 -17361.201,E2 -17361.201} C_VEL
LIN {X 0,Y 275.299,Z 469.31,A -85,B 0,C 180,E1 -17364.137,E2 -17364.137} C_VEL
LIN {X 0,Y 275.282,Z 470.187,A -85,B 0,C 180,E1 -17365.605,E2 -17365.605} C_VEL
LIN {X 0,Y 275.354,Z 470.635,A -85,B 0,C 180,E1 -17367.071,E2 -17367.071} C_VEL
LIN {X 0,Y 275.35,Z 470.692,A -85,B 0,C 180,E1 -17368.535,E2 -17368.535} C_VEL
LIN {X 0,Y 275.414,Z 470.364,A -85,B 0,C 180,E1 -17369.997,E2 -17369.997} C_VEL
LIN {X 0,Y 275.383,Z 469.634,A -85,B 0,C 180,E1 -17371.459,E2 -17371.459} C_VEL
LIN {X 0,Y 275.39,Z 468.455,A -85,B 0,C 180,E1 -17372.923,E2 -17372.923} C_VEL
LIN {X 0,Y 275.378,Z 465.294,A -85,B 0,C 180,E1 -17375.539,E2 -17375.539} C_VEL
LIN {X 0,Y 275.581,Z 460.879,A -85,B 0,C 180,E1 -17378.06,E2 -17378.06} C_VEL
LIN {X 0,Y 276.058,Z 454.781,A -85,B 0,C 180,E1 -17380.632,E2 -17380.632} C_VEL
LIN {X 0,Y 276.851,Z 448.081,A -85,B 0,C 180,E1 -17382.83,E2 -17382.83} C_VEL
LIN {X 0,Y 277.966,Z 439.75,A -85,B 0,C 180,E1 -17385.016,E2 -17385.016} C_VEL
LIN {X 0,Y 279.175,Z 430.611,A -85,B 0,C 180,E1 -17386.938,E2 -17386.938} C_VEL
LIN {X 0,Y 280.578,Z 420.625,A -85,B 0,C 180,E1 -17388.62,E2 -17388.62} C_VEL
LIN {X 0,Y 281.946,Z 410.147,A -85,B 0,C 180,E1 -17390.039,E2 -17390.039} C_VEL
LIN {X 0,Y 283.356,Z 398.654,A -85,B 0,C 180,E1 -17391.263,E2 -17391.263} C_VEL
LIN {X 0,Y 284.56,Z 386.785,A -85,B 0,C 180,E1 -17392.216,E2 -17392.216} C_VEL
LIN {X 0,Y 285.681,Z 373.098,A -85,B 0,C 180,E1 -17392.983,E2 -17392.983} C_VEL
LIN {X 0,Y 286.215,Z 360.13,A -85,B 0,C 180,E1 -17393.434,E2 -17393.434} C_VEL
LIN {X 0,Y 287.431,Z 304.59,A -85,B 0,C 180,E1 -17394.804,E2 -17394.804} C_VEL
LIN {X 0,Y 282.359,Z 264.52,A -85,B 0,C 180,E1 -17396.267,E2 -17396.267} C_VEL
LIN {X 0,Y 281.386,Z 257.528,A -85,B 0,C 180,E1 -17396.562,E2 -17396.562} C_VEL
LIN {X 0,Y 281.28,Z 254.213,A -85,B 0,C 180,E1 -17397.526,E2 -17397.526} C_VEL
LIN {X 0,Y 278.962,Z 242.821,A -85,B 0,C 180,E1 -17401.066,E2 -17401.066} C_VEL
LIN {X 0,Y 277.28,Z 234.95,A -85,B 0,C 180,E1 -17403.641,E2 -17403.641} C_VEL
LIN {X 0,Y 277.253,Z 234.951,A -85,B 0,C 180,E1 -17407.464,E2 -17407.464} C_VEL
LIN {X 0,Y 277.189,Z 234.956,A -85,B 0,C 180,E1 -17411.232,E2 -17411.232} C_VEL
LIN {X 0,Y 277.207,Z 234.954,A -85,B 0,C 180,E1 -17415.216,E2 -17415.216} C_VEL
LIN {X 0,Y 277.267,Z 234.949,A -85,B 0,C 180,E1 -17419.491,E2 -17419.491} C_VEL
LIN {X 0,Y 277.249,Z 234.948,A -85,B 0,C 180,E1 -17422.528,E2 -17422.528} C_VEL
LIN {X 0,Y 277.217,Z 234.952,A -85,B 0,C 180,E1 -17426.1,E2 -17426.1} C_VEL
LIN {X 0,Y 277.23,Z 234.953,A -85,B 0,C 180,E1 -17429.535,E2 -17429.535} C_VEL
LIN {X 0,Y 277.324,Z 234.938,A -85,B 0,C 180,E1 -17432.86,E2 -17432.86} C_VEL
LIN {X 0,Y 277.341,Z 234.936,A -85,B 0,C 180,E1 -17436.081,E2 -17436.081} C_VEL
LIN {X 0,Y 277.333,Z 234.937,A -85,B 0,C 180,E1 -17440.765,E2 -17440.765} C_VEL
LIN {X 0,Y 277.376,Z 234.934,A -85,B 0,C 180,E1 -17445.323,E2 -17445.323} C_VEL
LIN {X 0,Y 277.423,Z 234.926,A -85,B 0,C 180,E1 -17449.786,E2 -17449.786} C_VEL
LIN {X 0,Y 277.608,Z 234.901,A -85,B 0,C 180,E1 -17452.728,E2 -17452.728} C_VEL
LIN {X 0,Y 277.777,Z 234.88,A -85,B 0,C 180,E1 -17458.55,E2 -17458.55} C_VEL
LIN {X 0,Y 277.776,Z 234.867,A -85,B 0,C 180,E1 -17461.45,E2 -17461.45} C_VEL
LIN {X 0,Y 277.592,Z 234.906,A -85,B 0,C 180,E1 -17467.273,E2 -17467.273} C_VEL
LIN {X 0,Y 277.419,Z 234.925,A -85,B 0,C 180,E1 -17470.215,E2 -17470.215} C_VEL
LIN {X 0,Y 277.369,Z 234.921,A -85,B 0,C 180,E1 -17474.678,E2 -17474.678} C_VEL
LIN {X 0,Y 277.247,Z 234.948,A -85,B 0,C 180,E1 -17479.241,E2 -17479.241} C_VEL
LIN {X 0,Y 277.26,Z 234.944,A -85,B 0,C 180,E1 -17483.927,E2 -17483.927} C_VEL
LIN {X 0,Y 277.288,Z 234.942,A -85,B 0,C 180,E1 -17487.507,E2 -17487.507} C_VEL
LIN {X 0,Y 277.242,Z 234.951,A -85,B 0,C 180,E1 -17490.485,E2 -17490.485} C_VEL
LIN {X 0,Y 277.218,Z 234.951,A -85,B 0,C 180,E1 -17493.9,E2 -17493.9} C_VEL
LIN {X 0,Y 277.255,Z 234.946,A -85,B 0,C 180,E1 -17497.472,E2 -17497.472} C_VEL
LIN {X 0,Y 277.233,Z 234.949,A -85,B 0,C 180,E1 -17501.233,E2 -17501.233} C_VEL
LIN {X 0,Y 277.201,Z 234.945,A -85,B 0,C 180,E1 -17505.227,E2 -17505.227} C_VEL
LIN {X 0,Y 277.203,Z 234.953,A -85,B 0,C 180,E1 -17509.517,E2 -17509.517} C_VEL
LIN {X 0,Y 277.247,Z 234.943,A -85,B 0,C 180,E1 -17512.535,E2 -17512.535} C_VEL
LIN {X 0,Y 277.232,Z 234.953,A -85,B 0,C 180,E1 -17516.109,E2 -17516.109} C_VEL
LIN {X 0,Y 277.25,Z 234.949,A -85,B 0,C 180,E1 -17519.544,E2 -17519.544} C_VEL
LIN {X 0,Y 277.348,Z 234.935,A -85,B 0,C 180,E1 -17522.869,E2 -17522.869} C_VEL
LIN {X 0,Y 277.289,Z 234.944,A -85,B 0,C 180,E1 -17526.081,E2 -17526.081} C_VEL
LIN {X 0,Y 277.306,Z 234.941,A -85,B 0,C 180,E1 -17530.768,E2 -17530.768} C_VEL
LIN {X 0,Y 277.388,Z 234.932,A -85,B 0,C 180,E1 -17534.214,E2 -17534.214} C_VEL
LIN {X 0,Y 278.48,Z 237.908,A -85,B 0,C 180,E1 -17534.403,E2 -17534.403} C_VEL
LIN {X 0,Y 282.782,Z 248.591,A -85,B 0,C 180,E1 -17535.058,E2 -17535.058} C_VEL
LIN {X 0,Y 288.331,Z 264.915,A -85,B 0,C 180,E1 -17535.94,E2 -17535.94} C_VEL
LIN {X 0,Y 286.31,Z 341.193,A -85,B 0,C 180,E1 -17537.826,E2 -17537.826} C_VEL
LIN {X 0,Y 285.55,Z 354.568,A -85,B 0,C 180,E1 -17538.423,E2 -17538.423} C_VEL
LIN {X 0,Y 284.736,Z 366.699,A -85,B 0,C 180,E1 -17539.246,E2 -17539.246} C_VEL
LIN {X 0,Y 283.919,Z 377.236,A -85,B 0,C 180,E1 -17540.205,E2 -17540.205} C_VEL
LIN {X 0,Y 282.63,Z 387.933,A -85,B 0,C 180,E1 -17541.423,E2 -17541.423} C_VEL
LIN {X 0,Y 281.36,Z 397.761,A -85,B 0,C 180,E1 -17542.829,E2 -17542.829} C_VEL
LIN {X 0,Y 279.93,Z 407.706,A -85,B 0,C 180,E1 -17544.601,E2 -17544.601} C_VEL
LIN {X 0,Y 278.632,Z 417.322,A -85,B 0,C 180,E1 -17546.75,E2 -17546.75} C_VEL
LIN {X 0,Y 277.437,Z 425.012,A -85,B 0,C 180,E1 -17548.914,E2 -17548.914} C_VEL
LIN {X 0,Y 276.573,Z 432.07,A -85,B 0,C 180,E1 -17551.459,E2 -17551.459} C_VEL
LIN {X 0,Y 275.989,Z 436.785,A -85,B 0,C 180,E1 -17553.652,E2 -17553.652} C_VEL
LIN {X 0,Y 275.678,Z 440.806,A -85,B 0,C 180,E1 -17556.144,E2 -17556.144} C_VEL
LIN {X 0,Y 275.332,Z 443.659,A -85,B 0,C 180,E1 -17558.812,E2 -17558.812} C_VEL
LIN {X 0,Y 275.281,Z 445.275,A -85,B 0,C 180,E1 -17561.787,E2 -17561.787} C_VEL
LIN {X 0,Y 275.553,Z 445.378,A -85,B 0,C 180,E1 -17564.258,E2 -17564.258} C_VEL
LIN {X 0,Y 275.804,Z 444.613,A -85,B 0,C 180,E1 -17566.279,E2 -17566.279} C_VEL
LIN {X 0,Y 276.189,Z 443.588,A -85,B 0,C 180,E1 -17567.781,E2 -17567.781} C_VEL
LIN {X 0,Y 277.097,Z 440.973,A -85,B 0,C 180,E1 -17570.209,E2 -17570.209} C_VEL
LIN {X 0,Y 278.044,Z 437.776,A -85,B 0,C 180,E1 -17572.282,E2 -17572.282} C_VEL
LIN {X 0,Y 279.399,Z 433.208,A -85,B 0,C 180,E1 -17574.522,E2 -17574.522} C_VEL
LIN {X 0,Y 281.092,Z 427.324,A -85,B 0,C 180,E1 -17576.747,E2 -17576.747} C_VEL
LIN {X 0,Y 283.143,Z 419.898,A -85,B 0,C 180,E1 -17578.948,E2 -17578.948} C_VEL
LIN {X 0,Y 285.189,Z 412.005,A -85,B 0,C 180,E1 -17580.822,E2 -17580.822} C_VEL
LIN {X 0,Y 287.288,Z 402.988,A -85,B 0,C 180,E1 -17582.56,E2 -17582.56} C_VEL
LIN {X 0,Y 289.573,Z 392.516,A -85,B 0,C 180,E1 -17584.155,E2 -17584.155} C_VEL
LIN {X 0,Y 291.608,Z 380.939,A -85,B 0,C 180,E1 -17585.55,E2 -17585.55} C_VEL
LIN {X 0,Y 293.272,Z 368.663,A -85,B 0,C 180,E1 -17586.698,E2 -17586.698} C_VEL
LIN {X 0,Y 294.74,Z 355.65,A -85,B 0,C 180,E1 -17587.555,E2 -17587.555} C_VEL
LIN {X 0,Y 295.685,Z 343.109,A -85,B 0,C 180,E1 -17588.114,E2 -17588.114} C_VEL
LIN {X 0,Y 297.543,Z 291.799,A -85,B 0,C 180,E1 -17589.384,E2 -17589.384} C_VEL
LIN {X 0,Y 298.082,Z 276.083,A -85,B 0,C 180,E1 -17589.762,E2 -17589.762} C_VEL
LIN {X 0,Y 291.24,Z 261.03,A -85,B 0,C 180,E1 -17591.091,E2 -17591.091} C_VEL
LIN {X 0,Y 283.39,Z 246.203,A -85,B 0,C 180,E1 -17592.653,E2 -17592.653} C_VEL
LIN {X 0,Y 279.09,Z 238.811,A -85,B 0,C 180,E1 -17593.538,E2 -17593.538} C_VEL
LIN {X 0,Y 277.636,Z 236.438,A -85,B 0,C 180,E1 -17593.842,E2 -17593.842} C_VEL
LIN {X 0,Y 277.387,Z 235.532,A -85,B 0,C 180,E1 -17593.976,E2 -17593.976} C_VEL
LIN {X 0,Y 277.271,Z 234.935,A -85,B 0,C 180,E1 -17594.231,E2 -17594.231} C_VEL
LIN {X 0,Y 277.287,Z 234.947,A -85,B 0,C 180,E1 -17598.777,E2 -17598.777} C_VEL
LIN {X 0,Y 277.27,Z 234.941,A -85,B 0,C 180,E1 -17602.531,E2 -17602.531} C_VEL
LIN {X 0,Y 277.239,Z 234.946,A -85,B 0,C 180,E1 -17606.103,E2 -17606.103} C_VEL
LIN {X 0,Y 277.238,Z 234.945,A -85,B 0,C 180,E1 -17610.47,E2 -17610.47} C_VEL
LIN {X 0,Y 277.347,Z 234.929,A -85,B 0,C 180,E1 -17612.863,E2 -17612.863} C_VEL
LIN {X 0,Y 277.244,Z 234.94,A -85,B 0,C 180,E1 -17616.762,E2 -17616.762} C_VEL
LIN {X 0,Y 276.552,Z 235.037,A -85,B 0,C 180,E1 -17617.974,E2 -17617.974} C_VEL
LIN {X 0,Y 273.684,Z 235.385,A -85,B 0,C 180,E1 -17619.949,E2 -17619.949} C_VEL
LIN {X 0,Y 271.297,Z 235.685,A -85,B 0,C 180,E1 -17621.555,E2 -17621.555} C_VEL
LIN {X 0,Y 270.321,Z 235.812,A -85,B 0,C 180,E1 -17622.799,E2 -17622.799} C_VEL
LIN {X 0,Y 270.266,Z 235.815,A -85,B 0,C 180,E1 -17623.22,E2 -17623.22} C_VEL
LIN {X 0,Y 270.331,Z 235.81,A -85,B 0,C 180,E1 -17626.468,E2 -17626.468} C_VEL
LIN {X 0,Y 270.535,Z 235.785,A -85,B 0,C 180,E1 -17631.033,E2 -17631.033} C_VEL
LIN {X 0,Y 270.517,Z 235.779,A -85,B 0,C 180,E1 -17634.035,E2 -17634.035} C_VEL
LIN {X 0,Y 270.767,Z 235.744,A -85,B 0,C 180,E1 -17638.513,E2 -17638.513} C_VEL
LIN {X 0,Y 270.765,Z 235.753,A -85,B 0,C 180,E1 -17641.487,E2 -17641.487} C_VEL
LIN {X 0,Y 270.538,Z 235.773,A -85,B 0,C 180,E1 -17647.463,E2 -17647.463} C_VEL
LIN {X 0,Y 270.372,Z 235.806,A -85,B 0,C 180,E1 -17650.484,E2 -17650.484} C_VEL
LIN {X 0,Y 270.353,Z 235.807,A -85,B 0,C 180,E1 -17655.067,E2 -17655.067} C_VEL
LIN {X 0,Y 270.209,Z 235.825,A -85,B 0,C 180,E1 -17659.763,E2 -17659.763} C_VEL
LIN {X 0,Y 270.172,Z 235.828,A -85,B 0,C 180,E1 -17664.437,E2 -17664.437} C_VEL
LIN {X 0,Y 270.174,Z 235.831,A -85,B 0,C 180,E1 -17667.92,E2 -17667.92} C_VEL
LIN {X 0,Y 270.154,Z 235.833,A -85,B 0,C 180,E1 -17671.352,E2 -17671.352} C_VEL
LIN {X 0,Y 270.186,Z 235.829,A -85,B 0,C 180,E1 -17674.908,E2 -17674.908} C_VEL
LIN {X 0,Y 270.192,Z 235.799,A -85,B 0,C 180,E1 -17678.711,E2 -17678.711} C_VEL
LIN {X 0,Y 270.155,Z 235.83,A -85,B 0,C 180,E1 -17683.249,E2 -17683.249} C_VEL
LIN {X 0,Y 270.146,Z 235.825,A -85,B 0,C 180,E1 -17687.438,E2 -17687.438} C_VEL
LIN {X 0,Y 270.153,Z 235.855,A -85,B 0,C 180,E1 -17688.847,E2 -17688.847} C_VEL
LIN {X 0,Y 272.961,Z 245.678,A -85,B 0,C 180,E1 -17692.955,E2 -17692.955} C_VEL
LIN {X 0,Y 275.102,Z 254.505,A -85,B 0,C 180,E1 -17696.332,E2 -17696.332} C_VEL
LIN {X 0,Y 275.445,Z 255.92,A -85,B 0,C 180,E1 -17696.855,E2 -17696.855} C_VEL
LIN {X 0,Y 277.629,Z 260.387,A -85,B 0,C 180,E1 -17697.338,E2 -17697.338} C_VEL
LIN {X 0,Y 285.252,Z 276.845,A -85,B 0,C 180,E1 -17698.97,E2 -17698.97} C_VEL
LIN {X 0,Y 287.289,Z 286.636,A -85,B 0,C 180,E1 -17699.547,E2 -17699.547} C_VEL
LIN {X 0,Y 290.868,Z 308.273,A -85,B 0,C 180,E1 -17700.66,E2 -17700.66} C_VEL
LIN {X 0,Y 290.782,Z 317.22,A -85,B 0,C 180,E1 -17700.909,E2 -17700.909} C_VEL
LIN {X 0,Y 288.974,Z 365.914,A -85,B 0,C 180,E1 -17702.135,E2 -17702.135} C_VEL
LIN {X 0,Y 287.679,Z 379.668,A -85,B 0,C 180,E1 -17702.738,E2 -17702.738} C_VEL
LIN {X 0,Y 285.999,Z 392.06,A -85,B 0,C 180,E1 -17703.551,E2 -17703.551} C_VEL
LIN {X 0,Y 284.107,Z 403.137,A -85,B 0,C 180,E1 -17704.544,E2 -17704.544} C_VEL
LIN {X 0,Y 281.715,Z 414.683,A -85,B 0,C 180,E1 -17705.888,E2 -17705.888} C_VEL
LIN {X 0,Y 279.298,Z 425.092,A -85,B 0,C 180,E1 -17707.434,E2 -17707.434} C_VEL
LIN {X 0,Y 276.954,Z 434.495,A -85,B 0,C 180,E1 -17709.19,E2 -17709.19} C_VEL
LIN {X 0,Y 274.665,Z 442.92,A -85,B 0,C 180,E1 -17711.156,E2 -17711.156} C_VEL
LIN {X 0,Y 272.579,Z 450.936,A -85,B 0,C 180,E1 -17713.523,E2 -17713.523} C_VEL
LIN {X 0,Y 270.927,Z 456.861,A -85,B 0,C 180,E1 -17715.732,E2 -17715.732} C_VEL
LIN {X 0,Y 269.65,Z 461.563,A -85,B 0,C 180,E1 -17717.963,E2 -17717.963} C_VEL
LIN {X 0,Y 268.889,Z 465.18,A -85,B 0,C 180,E1 -17720.217,E2 -17720.217} C_VEL
LIN {X 0,Y 268.381,Z 467.806,A -85,B 0,C 180,E1 -17722.474,E2 -17722.474} C_VEL
LIN {X 0,Y 268.221,Z 469.476,A -85,B 0,C 180,E1 -17724.677,E2 -17724.677} C_VEL
LIN {X 0,Y 268.258,Z 470.318,A -85,B 0,C 180,E1 -17726.994,E2 -17726.994} C_VEL
LIN {X 0,Y 268.273,Z 470.354,A -85,B 0,C 180,E1 -17728.496,E2 -17728.496} C_VEL
LIN {X 0,Y 268.331,Z 470.003,A -85,B 0,C 180,E1 -17729.997,E2 -17729.997} C_VEL
LIN {X 0,Y 268.305,Z 469.235,A -85,B 0,C 180,E1 -17731.498,E2 -17731.498} C_VEL
LIN {X 0,Y 268.317,Z 468.026,A -85,B 0,C 180,E1 -17733,E2 -17733} C_VEL
LIN {X 0,Y 268.278,Z 465.148,A -85,B 0,C 180,E1 -17735.452,E2 -17735.452} C_VEL
LIN {X 0,Y 268.436,Z 461.793,A -85,B 0,C 180,E1 -17737.518,E2 -17737.518} C_VEL
LIN {X 0,Y 268.773,Z 457.019,A -85,B 0,C 180,E1 -17739.782,E2 -17739.782} C_VEL
LIN {X 0,Y 269.541,Z 449.833,A -85,B 0,C 180,E1 -17742.418,E2 -17742.418} C_VEL
LIN {X 0,Y 270.631,Z 442.008,A -85,B 0,C 180,E1 -17744.662,E2 -17744.662} C_VEL
LIN {X 0,Y 271.722,Z 433.978,A -85,B 0,C 180,E1 -17746.525,E2 -17746.525} C_VEL
LIN {X 0,Y 273.184,Z 424.185,A -85,B 0,C 180,E1 -17748.365,E2 -17748.365} C_VEL
LIN {X 0,Y 274.648,Z 413.283,A -85,B 0,C 180,E1 -17750.009,E2 -17750.009} C_VEL
LIN {X 0,Y 276.1,Z 402.672,A -85,B 0,C 180,E1 -17751.263,E2 -17751.263} C_VEL
LIN {X 0,Y 277.536,Z 389.865,A -85,B 0,C 180,E1 -17752.417,E2 -17752.417} C_VEL
LIN {X 0,Y 278.664,Z 377.031,A -85,B 0,C 180,E1 -17753.252,E2 -17753.252} C_VEL
LIN {X 0,Y 279.421,Z 363.962,A -85,B 0,C 180,E1 -17753.795,E2 -17753.795} C_VEL
LIN {X 0,Y 280.728,Z 304.819,A -85,B 0,C 180,E1 -17755.309,E2 -17755.309} C_VEL
LIN {X 0,Y 275.727,Z 265.022,A -85,B 0,C 180,E1 -17756.805,E2 -17756.805} C_VEL
LIN {X 0,Y 274.538,Z 257.211,A -85,B 0,C 180,E1 -17757.148,E2 -17757.148} C_VEL
LIN {X 0,Y 272.475,Z 246.221,A -85,B 0,C 180,E1 -17760.618,E2 -17760.618} C_VEL
LIN {X 0,Y 270.203,Z 235.833,A -85,B 0,C 180,E1 -17764.135,E2 -17764.135} C_VEL
LIN {X 0,Y 270.21,Z 235.828,A -85,B 0,C 180,E1 -17766.735,E2 -17766.735} C_VEL
LIN {X 0,Y 270.149,Z 235.833,A -85,B 0,C 180,E1 -17771.023,E2 -17771.023} C_VEL
LIN {X 0,Y 270.157,Z 235.833,A -85,B 0,C 180,E1 -17775.381,E2 -17775.381} C_VEL
LIN {X 0,Y 270.218,Z 235.827,A -85,B 0,C 180,E1 -17779.442,E2 -17779.442} C_VEL
LIN {X 0,Y 270.217,Z 235.827,A -85,B 0,C 180,E1 -17783.721,E2 -17783.721} C_VEL
LIN {X 0,Y 270.172,Z 235.829,A -85,B 0,C 180,E1 -17786.888,E2 -17786.888} C_VEL
LIN {X 0,Y 270.196,Z 235.826,A -85,B 0,C 180,E1 -17790.383,E2 -17790.383} C_VEL
LIN {X 0,Y 270.234,Z 235.824,A -85,B 0,C 180,E1 -17793.761,E2 -17793.761} C_VEL
LIN {X 0,Y 270.236,Z 235.822,A -85,B 0,C 180,E1 -17797.039,E2 -17797.039} C_VEL
LIN {X 0,Y 270.291,Z 235.814,A -85,B 0,C 180,E1 -17800.244,E2 -17800.244} C_VEL
LIN {X 0,Y 270.343,Z 235.81,A -85,B 0,C 180,E1 -17804.932,E2 -17804.932} C_VEL
LIN {X 0,Y 270.374,Z 235.806,A -85,B 0,C 180,E1 -17809.516,E2 -17809.516} C_VEL
LIN {X 0,Y 270.567,Z 235.777,A -85,B 0,C 180,E1 -17812.538,E2 -17812.538} C_VEL
LIN {X 0,Y 270.743,Z 235.756,A -85,B 0,C 180,E1 -17818.513,E2 -17818.513} C_VEL
LIN {X 0,Y 270.742,Z 235.742,A -85,B 0,C 180,E1 -17821.488,E2 -17821.488} C_VEL
LIN {X 0,Y 270.549,Z 235.782,A -85,B 0,C 180,E1 -17827.463,E2 -17827.463} C_VEL
LIN {X 0,Y 270.372,Z 235.804,A -85,B 0,C 180,E1 -17830.484,E2 -17830.484} C_VEL
LIN {X 0,Y 270.328,Z 235.798,A -85,B 0,C 180,E1 -17835.069,E2 -17835.069} C_VEL
LIN {X 0,Y 270.186,Z 235.827,A -85,B 0,C 180,E1 -17839.765,E2 -17839.765} C_VEL
LIN {X 0,Y 270.203,Z 235.827,A -85,B 0,C 180,E1 -17844.593,E2 -17844.593} C_VEL
LIN {X 0,Y 270.238,Z 235.821,A -85,B 0,C 180,E1 -17847.913,E2 -17847.913} C_VEL
LIN {X 0,Y 270.154,Z 235.831,A -85,B 0,C 180,E1 -17851.352,E2 -17851.352} C_VEL
LIN {X 0,Y 270.177,Z 235.829,A -85,B 0,C 180,E1 -17854.91,E2 -17854.91} C_VEL
LIN {X 0,Y 270.197,Z 235.824,A -85,B 0,C 180,E1 -17858.722,E2 -17858.722} C_VEL
LIN {X 0,Y 270.189,Z 235.827,A -85,B 0,C 180,E1 -17862.555,E2 -17862.555} C_VEL
LIN {X 0,Y 270.151,Z 235.827,A -85,B 0,C 180,E1 -17866.755,E2 -17866.755} C_VEL
LIN {X 0,Y 270.19,Z 235.825,A -85,B 0,C 180,E1 -17871.379,E2 -17871.379} C_VEL
LIN {X 0,Y 270.186,Z 235.827,A -85,B 0,C 180,E1 -17875.1,E2 -17875.1} C_VEL
LIN {X 0,Y 270.188,Z 235.827,A -85,B 0,C 180,E1 -17879.136,E2 -17879.136} C_VEL
LIN {X 0,Y 270.253,Z 235.822,A -85,B 0,C 180,E1 -17882.151,E2 -17882.151} C_VEL
LIN {X 0,Y 270.229,Z 235.822,A -85,B 0,C 180,E1 -17885.543,E2 -17885.543} C_VEL
LIN {X 0,Y 270.249,Z 235.821,A -85,B 0,C 180,E1 -17890.246,E2 -17890.246} C_VEL
LIN {X 0,Y 270.314,Z 235.863,A -85,B 0,C 180,E1 -17893.616,E2 -17893.616} C_VEL
LIN {X 0,Y 271.457,Z 238.886,A -85,B 0,C 180,E1 -17893.806,E2 -17893.806} C_VEL
LIN {X 0,Y 275.607,Z 248.538,A -85,B 0,C 180,E1 -17894.448,E2 -17894.448} C_VEL
LIN {X 0,Y 281.66,Z 265.989,A -85,B 0,C 180,E1 -17895.438,E2 -17895.438} C_VEL
LIN {X 0,Y 279.633,Z 341.432,A -85,B 0,C 180,E1 -17897.346,E2 -17897.346} C_VEL
LIN {X 0,Y 278.849,Z 354.842,A -85,B 0,C 180,E1 -17897.957,E2 -17897.957} C_VEL
LIN {X 0,Y 278.003,Z 366.988,A -85,B 0,C 180,E1 -17898.798,E2 -17898.798} C_VEL
LIN {X 0,Y 277.139,Z 377.539,A -85,B 0,C 180,E1 -17899.779,E2 -17899.779} C_VEL
LIN {X 0,Y 275.821,Z 388.238,A -85,B 0,C 180,E1 -17901.025,E2 -17901.025} C_VEL
LIN {X 0,Y 274.503,Z 398.07,A -85,B 0,C 180,E1 -17902.464,E2 -17902.464} C_VEL
LIN {X 0,Y 273.171,Z 407.129,A -85,B 0,C 180,E1 -17904.097,E2 -17904.097} C_VEL
LIN {X 0,Y 271.973,Z 415.42,A -85,B 0,C 180,E1 -17905.928,E2 -17905.928} C_VEL
LIN {X 0,Y 270.744,Z 423.544,A -85,B 0,C 180,E1 -17908.144,E2 -17908.144} C_VEL
LIN {X 0,Y 269.881,Z 429.086,A -85,B 0,C 180,E1 -17910.003,E2 -17910.003} C_VEL
LIN {X 0,Y 269.28,Z 434.486,A -85,B 0,C 180,E1 -17912.246,E2 -17912.246} C_VEL
LIN {X 0,Y 268.821,Z 438.724,A -85,B 0,C 180,E1 -17914.501,E2 -17914.501} C_VEL
LIN {X 0,Y 268.597,Z 441.132,A -85,B 0,C 180,E1 -17916.121,E2 -17916.121} C_VEL
LIN {X 0,Y 268.225,Z 444.129,A -85,B 0,C 180,E1 -17919.047,E2 -17919.047} C_VEL
LIN {X 0,Y 268.145,Z 445.094,A -85,B 0,C 180,E1 -17920.574,E2 -17920.574} C_VEL
LIN {X 0,Y 268.215,Z 445.659,A -85,B 0,C 180,E1 -17922.102,E2 -17922.102} C_VEL
LIN {X 0,Y 268.49,Z 445.711,A -85,B 0,C 180,E1 -17924.415,E2 -17924.415} C_VEL
LIN {X 0,Y 268.829,Z 444.846,A -85,B 0,C 180,E1 -17926.714,E2 -17926.714} C_VEL
LIN {X 0,Y 269.243,Z 443.758,A -85,B 0,C 180,E1 -17928.255,E2 -17928.255} C_VEL
LIN {X 0,Y 270.113,Z 441.378,A -85,B 0,C 180,E1 -17930.498,E2 -17930.498} C_VEL
LIN {X 0,Y 271.247,Z 437.781,A -85,B 0,C 180,E1 -17932.871,E2 -17932.871} C_VEL
LIN {X 0,Y 272.674,Z 433.279,A -85,B 0,C 180,E1 -17935.089,E2 -17935.089} C_VEL
LIN {X 0,Y 274.563,Z 427.1,A -85,B 0,C 180,E1 -17937.436,E2 -17937.436} C_VEL
LIN {X 0,Y 276.761,Z 419.558,A -85,B 0,C 180,E1 -17939.681,E2 -17939.681} C_VEL
LIN {X 0,Y 278.789,Z 411.921,A -85,B 0,C 180,E1 -17941.51,E2 -17941.51} C_VEL
LIN {X 0,Y 281.112,Z 402.305,A -85,B 0,C 180,E1 -17943.368,E2 -17943.368} C_VEL
LIN {X 0,Y 283.555,Z 391.54,A -85,B 0,C 180,E1 -17944.988,E2 -17944.988} C_VEL
LIN {X 0,Y 285.668,Z 379.687,A -85,B 0,C 180,E1 -17946.407,E2 -17946.407} C_VEL
LIN {X 0,Y 287.301,Z 367.916,A -85,B 0,C 180,E1 -17947.48,E2 -17947.48} C_VEL
LIN {X 0,Y 288.813,Z 354.511,A -85,B 0,C 180,E1 -17948.353,E2 -17948.353} C_VEL
LIN {X 0,Y 289.73,Z 342.418,A -85,B 0,C 180,E1 -17948.876,E2 -17948.876} C_VEL
LIN {X 0,Y 292.019,Z 277.962,A -85,B 0,C 180,E1 -17950.489,E2 -17950.489} C_VEL
LIN {X 0,Y 285.217,Z 263.089,A -85,B 0,C 180,E1 -17951.868,E2 -17951.868} C_VEL
LIN {X 0,Y 277.038,Z 247.786,A -85,B 0,C 180,E1 -17953.572,E2 -17953.572} C_VEL
LIN {X 0,Y 274.154,Z 243.111,A -85,B 0,C 180,E1 -17954.183,E2 -17954.183} C_VEL
LIN {X 0,Y 272.198,Z 239.887,A -85,B 0,C 180,E1 -17954.61,E2 -17954.61} C_VEL
LIN {X 0,Y 270.564,Z 237.344,A -85,B 0,C 180,E1 -17954.97,E2 -17954.97} C_VEL
LIN {X 0,Y 270.267,Z 236.111,A -85,B 0,C 180,E1 -17955.073,E2 -17955.073} C_VEL
LIN {X 0,Y 270.194,Z 235.825,A -85,B 0,C 180,E1 -17955.388,E2 -17955.388} C_VEL
LIN {X 0,Y 270.244,Z 235.82,A -85,B 0,C 180,E1 -17959.446,E2 -17959.446} C_VEL
LIN {X 0,Y 270.237,Z 235.822,A -85,B 0,C 180,E1 -17963.724,E2 -17963.724} C_VEL
LIN {X 0,Y 270.195,Z 235.828,A -85,B 0,C 180,E1 -17966.891,E2 -17966.891} C_VEL
LIN {X 0,Y 270.22,Z 235.826,A -85,B 0,C 180,E1 -17970.385,E2 -17970.385} C_VEL
LIN {X 0,Y 270.25,Z 235.818,A -85,B 0,C 180,E1 -17973.762,E2 -17973.762} C_VEL
LIN {X 0,Y 270.194,Z 235.82,A -85,B 0,C 180,E1 -17977.035,E2 -17977.035} C_VEL
LIN {X 0,Y 270.249,Z 235.811,A -85,B 0,C 180,E1 -17980.24,E2 -17980.24} C_VEL
LIN {X 0,Y 270.266,Z 235.815,A -85,B 0,C 180,E1 -17983.22,E2 -17983.22} C_VEL
LIN {X 0,Y 269.656,Z 235.896,A -85,B 0,C 180,E1 -17984.464,E2 -17984.464} C_VEL
LIN {X 0,Y 266.807,Z 236.249,A -85,B 0,C 180,E1 -17986.492,E2 -17986.492} C_VEL
LIN {X 0,Y 264.391,Z 236.546,A -85,B 0,C 180,E1 -17988.142,E2 -17988.142} C_VEL
LIN {X 0,Y 263.406,Z 236.664,A -85,B 0,C 180,E1 -17989.421,E2 -17989.421} C_VEL
LIN {X 0,Y 263.357,Z 236.671,A -85,B 0,C 180,E1 -17989.854,E2 -17989.854} C_VEL
LIN {X 0,Y 263.538,Z 236.655,A -85,B 0,C 180,E1 -17992.337,E2 -17992.337} C_VEL
LIN {X 0,Y 263.732,Z 236.621,A -85,B 0,C 180,E1 -17998.473,E2 -17998.473} C_VEL
LIN {X 0,Y 263.728,Z 236.63,A -85,B 0,C 180,E1 -18001.527,E2 -18001.527} C_VEL
LIN {X 0,Y 263.5,Z 236.649,A -85,B 0,C 180,E1 -18007.664,E2 -18007.664} C_VEL
LIN {X 0,Y 263.318,Z 236.682,A -85,B 0,C 180,E1 -18010.768,E2 -18010.768} C_VEL
LIN {X 0,Y 263.296,Z 236.684,A -85,B 0,C 180,E1 -18015.481,E2 -18015.481} C_VEL
LIN {X 0,Y 263.195,Z 236.695,A -85,B 0,C 180,E1 -18020.312,E2 -18020.312} C_VEL
LIN {X 0,Y 263.113,Z 236.704,A -85,B 0,C 180,E1 -18024.751,E2 -18024.751} C_VEL
LIN {X 0,Y 263.107,Z 236.706,A -85,B 0,C 180,E1 -18028.738,E2 -18028.738} C_VEL
LIN {X 0,Y 263.108,Z 236.709,A -85,B 0,C 180,E1 -18032.292,E2 -18032.292} C_VEL
LIN {X 0,Y 263.148,Z 236.702,A -85,B 0,C 180,E1 -18035.984,E2 -18035.984} C_VEL
LIN {X 0,Y 263.097,Z 236.691,A -85,B 0,C 180,E1 -18039.874,E2 -18039.874} C_VEL
LIN {X 0,Y 263.097,Z 236.714,A -85,B 0,C 180,E1 -18043.99,E2 -18043.99} C_VEL
LIN {X 0,Y 263.125,Z 236.882,A -85,B 0,C 180,E1 -18047.855,E2 -18047.855} C_VEL
LIN {X 0,Y 265.783,Z 246.049,A -85,B 0,C 180,E1 -18051.875,E2 -18051.875} C_VEL
LIN {X 0,Y 268.084,Z 255.156,A -85,B 0,C 180,E1 -18055.523,E2 -18055.523} C_VEL
LIN {X 0,Y 268.329,Z 255.968,A -85,B 0,C 180,E1 -18055.693,E2 -18055.693} C_VEL
LIN {X 0,Y 275.601,Z 270.666,A -85,B 0,C 180,E1 -18057.353,E2 -18057.353} C_VEL
LIN {X 0,Y 280.042,Z 280.613,A -85,B 0,C 180,E1 -18058.337,E2 -18058.337} C_VEL
LIN {X 0,Y 284.239,Z 304.401,A -85,B 0,C 180,E1 -18059.663,E2 -18059.663} C_VEL
LIN {X 0,Y 285.076,Z 311.095,A -85,B 0,C 180,E1 -18059.978,E2 -18059.978} C_VEL
LIN {X 0,Y 283.012,Z 365.485,A -85,B 0,C 180,E1 -18061.372,E2 -18061.372} C_VEL
LIN {X 0,Y 281.73,Z 378.846,A -85,B 0,C 180,E1 -18061.961,E2 -18061.961} C_VEL
LIN {X 0,Y 279.876,Z 391.918,A -85,B 0,C 180,E1 -18062.825,E2 -18062.825} C_VEL
LIN {X 0,Y 277.732,Z 403.737,A -85,B 0,C 180,E1 -18063.917,E2 -18063.917} C_VEL
LIN {X 0,Y 275.277,Z 415.112,A -85,B 0,C 180,E1 -18065.287,E2 -18065.287} C_VEL
LIN {X 0,Y 272.764,Z 425.392,A -85,B 0,C 180,E1 -18066.863,E2 -18066.863} C_VEL
LIN {X 0,Y 270.331,Z 434.649,A -85,B 0,C 180,E1 -18068.655,E2 -18068.655} C_VEL
LIN {X 0,Y 268.027,Z 442.612,A -85,B 0,C 180,E1 -18070.56,E2 -18070.56} C_VEL
LIN {X 0,Y 266.048,Z 449.816,A -85,B 0,C 180,E1 -18072.71,E2 -18072.71} C_VEL
LIN {X 0,Y 264.597,Z 454.978,A -85,B 0,C 180,E1 -18074.595,E2 -18074.595} C_VEL
LIN {X 0,Y 263.067,Z 460.003,A -85,B 0,C 180,E1 -18076.873,E2 -18076.873} C_VEL
LIN {X 0,Y 262.087,Z 463.922,A -85,B 0,C 180,E1 -18079.179,E2 -18079.179} C_VEL
LIN {X 0,Y 261.668,Z 465.956,A -85,B 0,C 180,E1 -18080.724,E2 -18080.724} C_VEL
LIN {X 0,Y 261.148,Z 468.807,A -85,B 0,C 180,E1 -18083.818,E2 -18083.818} C_VEL
LIN {X 0,Y 261.165,Z 470.002,A -85,B 0,C 180,E1 -18086.912,E2 -18086.912} C_VEL
LIN {X 0,Y 261.197,Z 470.016,A -85,B 0,C 180,E1 -18088.455,E2 -18088.455} C_VEL
LIN {X 0,Y 261.251,Z 469.642,A -85,B 0,C 180,E1 -18089.997,E2 -18089.997} C_VEL
LIN {X 0,Y 261.228,Z 468.829,A -85,B 0,C 180,E1 -18091.539,E2 -18091.539} C_VEL
LIN {X 0,Y 261.222,Z 467.595,A -85,B 0,C 180,E1 -18093.081,E2 -18093.081} C_VEL
LIN {X 0,Y 261.189,Z 464.969,A -85,B 0,C 180,E1 -18095.384,E2 -18095.384} C_VEL
LIN {X 0,Y 261.358,Z 461.26,A -85,B 0,C 180,E1 -18097.723,E2 -18097.723} C_VEL
LIN {X 0,Y 261.722,Z 456.431,A -85,B 0,C 180,E1 -18100.048,E2 -18100.048} C_VEL
LIN {X 0,Y 262.379,Z 450.315,A -85,B 0,C 180,E1 -18102.369,E2 -18102.369} C_VEL
LIN {X 0,Y 263.536,Z 442.708,A -85,B 0,C 180,E1 -18104.671,E2 -18104.671} C_VEL
LIN {X 0,Y 264.66,Z 434.916,A -85,B 0,C 180,E1 -18106.582,E2 -18106.582} C_VEL
LIN {X 0,Y 266.081,Z 425.401,A -85,B 0,C 180,E1 -18108.474,E2 -18108.474} C_VEL
LIN {X 0,Y 267.593,Z 414.819,A -85,B 0,C 180,E1 -18110.159,E2 -18110.159} C_VEL
LIN {X 0,Y 269.246,Z 403.062,A -85,B 0,C 180,E1 -18111.63,E2 -18111.63} C_VEL
LIN {X 0,Y 270.692,Z 390.486,A -85,B 0,C 180,E1 -18112.814,E2 -18112.814} C_VEL
LIN {X 0,Y 271.938,Z 377.22,A -85,B 0,C 180,E1 -18113.71,E2 -18113.71} C_VEL
LIN {X 0,Y 272.705,Z 365.229,A -85,B 0,C 180,E1 -18114.245,E2 -18114.245} C_VEL
LIN {X 0,Y 274.09,Z 305.462,A -85,B 0,C 180,E1 -18115.819,E2 -18115.819} C_VEL
LIN {X 0,Y 269.226,Z 266.309,A -85,B 0,C 180,E1 -18117.336,E2 -18117.336} C_VEL
LIN {X 0,Y 267.839,Z 258.582,A -85,B 0,C 180,E1 -18117.683,E2 -18117.683} C_VEL
LIN {X 0,Y 267.379,Z 256.835,A -85,B 0,C 180,E1 -18117.808,E2 -18117.808} C_VEL
LIN {X 0,Y 265.328,Z 246.794,A -85,B 0,C 180,E1 -18121.092,E2 -18121.092} C_VEL
LIN {X 0,Y 263.17,Z 236.707,A -85,B 0,C 180,E1 -18124.567,E2 -18124.567} C_VEL
LIN {X 0,Y 263.145,Z 236.709,A -85,B 0,C 180,E1 -18127.891,E2 -18127.891} C_VEL
LIN {X 0,Y 263.104,Z 236.714,A -85,B 0,C 180,E1 -18131.888,E2 -18131.888} C_VEL
LIN {X 0,Y 263.118,Z 236.711,A -85,B 0,C 180,E1 -18136.142,E2 -18136.142} C_VEL
LIN {X 0,Y 263.133,Z 236.708,A -85,B 0,C 180,E1 -18140.132,E2 -18140.132} C_VEL
LIN {X 0,Y 263.15,Z 236.707,A -85,B 0,C 180,E1 -18144.016,E2 -18144.016} C_VEL
LIN {X 0,Y 263.102,Z 236.714,A -85,B 0,C 180,E1 -18147.708,E2 -18147.708} C_VEL
LIN {X 0,Y 263.169,Z 236.704,A -85,B 0,C 180,E1 -18151.78,E2 -18151.78} C_VEL
LIN {X 0,Y 263.186,Z 236.699,A -85,B 0,C 180,E1 -18156.387,E2 -18156.387} C_VEL
LIN {X 0,Y 263.254,Z 236.693,A -85,B 0,C 180,E1 -18159.693,E2 -18159.693} C_VEL
LIN {X 0,Y 263.291,Z 236.686,A -85,B 0,C 180,E1 -18164.518,E2 -18164.518} C_VEL
LIN {X 0,Y 263.316,Z 236.687,A -85,B 0,C 180,E1 -18169.232,E2 -18169.232} C_VEL
LIN {X 0,Y 263.526,Z 236.654,A -85,B 0,C 180,E1 -18172.337,E2 -18172.337} C_VEL
LIN {X 0,Y 263.708,Z 236.632,A -85,B 0,C 180,E1 -18178.473,E2 -18178.473} C_VEL
LIN {X 0,Y 263.706,Z 236.616,A -85,B 0,C 180,E1 -18181.527,E2 -18181.527} C_VEL
LIN {X 0,Y 263.511,Z 236.658,A -85,B 0,C 180,E1 -18187.664,E2 -18187.664} C_VEL
LIN {X 0,Y 263.311,Z 236.683,A -85,B 0,C 180,E1 -18190.768,E2 -18190.768} C_VEL
LIN {X 0,Y 263.271,Z 236.678,A -85,B 0,C 180,E1 -18195.483,E2 -18195.483} C_VEL
LIN {X 0,Y 263.173,Z 236.702,A -85,B 0,C 180,E1 -18200.314,E2 -18200.314} C_VEL
LIN {X 0,Y 263.158,Z 236.703,A -85,B 0,C 180,E1 -18205.297,E2 -18205.297} C_VEL
LIN {X 0,Y 263.134,Z 236.705,A -85,B 0,C 180,E1 -18208.735,E2 -18208.735} C_VEL
LIN {X 0,Y 263.103,Z 236.713,A -85,B 0,C 180,E1 -18212.293,E2 -18212.293} C_VEL
LIN {X 0,Y 263.172,Z 236.703,A -85,B 0,C 180,E1 -18216.772,E2 -18216.772} C_VEL
LIN {X 0,Y 263.133,Z 236.703,A -85,B 0,C 180,E1 -18219.868,E2 -18219.868} C_VEL
LIN {X 0,Y 263.117,Z 236.706,A -85,B 0,C 180,E1 -18223.986,E2 -18223.986} C_VEL
LIN {X 0,Y 263.105,Z 236.711,A -85,B 0,C 180,E1 -18228.412,E2 -18228.412} C_VEL
LIN {X 0,Y 263.165,Z 236.694,A -85,B 0,C 180,E1 -18233.243,E2 -18233.243} C_VEL
LIN {X 0,Y 263.119,Z 236.709,A -85,B 0,C 180,E1 -18237.717,E2 -18237.717} C_VEL
LIN {X 0,Y 263.186,Z 236.703,A -85,B 0,C 180,E1 -18241.79,E2 -18241.79} C_VEL
LIN {X 0,Y 263.193,Z 236.697,A -85,B 0,C 180,E1 -18245.217,E2 -18245.217} C_VEL
LIN {X 0,Y 263.231,Z 236.695,A -85,B 0,C 180,E1 -18249.696,E2 -18249.696} C_VEL
LIN {X 0,Y 263.209,Z 236.699,A -85,B 0,C 180,E1 -18252.963,E2 -18252.963} C_VEL
LIN {X 0,Y 264.341,Z 239.7,A -85,B 0,C 180,E1 -18253.163,E2 -18253.163} C_VEL
LIN {X 0,Y 269.163,Z 250.496,A -85,B 0,C 180,E1 -18253.928,E2 -18253.928} C_VEL
LIN {X 0,Y 275.068,Z 267.432,A -85,B 0,C 180,E1 -18254.929,E2 -18254.929} C_VEL
LIN {X 0,Y 272.976,Z 341.573,A -85,B 0,C 180,E1 -18256.843,E2 -18256.843} C_VEL
LIN {X 0,Y 272.167,Z 355.061,A -85,B 0,C 180,E1 -18257.467,E2 -18257.467} C_VEL
LIN {X 0,Y 271.289,Z 367.233,A -85,B 0,C 180,E1 -18258.327,E2 -18258.327} C_VEL
LIN {X 0,Y 270.231,Z 379.512,A -85,B 0,C 180,E1 -18259.515,E2 -18259.515} C_VEL
LIN {X 0,Y 268.638,Z 391.138,A -85,B 0,C 180,E1 -18260.973,E2 -18260.973} C_VEL
LIN {X 0,Y 267.179,Z 401.56,A -85,B 0,C 180,E1 -18262.636,E2 -18262.636} C_VEL
LIN {X 0,Y 265.828,Z 410.096,A -85,B 0,C 180,E1 -18264.314,E2 -18264.314} C_VEL
LIN {X 0,Y 264.711,Z 417.941,A -85,B 0,C 180,E1 -18266.197,E2 -18266.197} C_VEL
LIN {X 0,Y 263.622,Z 424.473,A -85,B 0,C 180,E1 -18268.093,E2 -18268.093} C_VEL
LIN {X 0,Y 262.794,Z 429.901,A -85,B 0,C 180,E1 -18270.003,E2 -18270.003} C_VEL
LIN {X 0,Y 262.173,Z 435.207,A -85,B 0,C 180,E1 -18272.307,E2 -18272.307} C_VEL
LIN {X 0,Y 261.732,Z 439.355,A -85,B 0,C 180,E1 -18274.623,E2 -18274.623} C_VEL
LIN {X 0,Y 261.495,Z 441.554,A -85,B 0,C 180,E1 -18276.174,E2 -18276.174} C_VEL
LIN {X 0,Y 261.251,Z 443.279,A -85,B 0,C 180,E1 -18277.732,E2 -18277.732} C_VEL
LIN {X 0,Y 261.119,Z 444.598,A -85,B 0,C 180,E1 -18279.295,E2 -18279.295} C_VEL
LIN {X 0,Y 261.052,Z 445.524,A -85,B 0,C 180,E1 -18280.864,E2 -18280.864} C_VEL
LIN {X 0,Y 261.167,Z 446.016,A -85,B 0,C 180,E1 -18282.434,E2 -18282.434} C_VEL
LIN {X 0,Y 261.424,Z 446.045,A -85,B 0,C 180,E1 -18284.576,E2 -18284.576} C_VEL
LIN {X 0,Y 261.841,Z 445.078,A -85,B 0,C 180,E1 -18287.174,E2 -18287.174} C_VEL
LIN {X 0,Y 262.328,Z 443.911,A -85,B 0,C 180,E1 -18288.754,E2 -18288.754} C_VEL
LIN {X 0,Y 263.144,Z 441.78,A -85,B 0,C 180,E1 -18290.807,E2 -18290.807} C_VEL
LIN {X 0,Y 264.524,Z 437.764,A -85,B 0,C 180,E1 -18293.487,E2 -18293.487} C_VEL
LIN {X 0,Y 266.391,Z 432.049,A -85,B 0,C 180,E1 -18296.233,E2 -18296.233} C_VEL
LIN {X 0,Y 268.427,Z 425.741,A -85,B 0,C 180,E1 -18298.544,E2 -18298.544} C_VEL
LIN {X 0,Y 270.843,Z 417.742,A -85,B 0,C 180,E1 -18300.829,E2 -18300.829} C_VEL
LIN {X 0,Y 273.053,Z 409.501,A -85,B 0,C 180,E1 -18302.718,E2 -18302.718} C_VEL
LIN {X 0,Y 275.558,Z 399.379,A -85,B 0,C 180,E1 -18304.574,E2 -18304.574} C_VEL
LIN {X 0,Y 277.857,Z 389.298,A -85,B 0,C 180,E1 -18306.027,E2 -18306.027} C_VEL
LIN {X 0,Y 279.757,Z 378.275,A -85,B 0,C 180,E1 -18307.304,E2 -18307.304} C_VEL
LIN {X 0,Y 281.393,Z 367.166,A -85,B 0,C 180,E1 -18308.294,E2 -18308.294} C_VEL
LIN {X 0,Y 282.857,Z 354.425,A -85,B 0,C 180,E1 -18309.123,E2 -18309.123} C_VEL
LIN {X 0,Y 283.762,Z 342.696,A -85,B 0,C 180,E1 -18309.634,E2 -18309.634} C_VEL
LIN {X 0,Y 286.109,Z 280.008,A -85,B 0,C 180,E1 -18311.229,E2 -18311.229} C_VEL
LIN {X 0,Y 278.645,Z 264.026,A -85,B 0,C 180,E1 -18312.807,E2 -18312.807} C_VEL
LIN {X 0,Y 270.368,Z 248.787,A -85,B 0,C 180,E1 -18314.62,E2 -18314.62} C_VEL
LIN {X 0,Y 265.914,Z 241.83,A -85,B 0,C 180,E1 -18315.622,E2 -18315.622} C_VEL
LIN {X 0,Y 263.683,Z 238.623,A -85,B 0,C 180,E1 -18316.133,E2 -18316.133} C_VEL
LIN {X 0,Y 263.153,Z 236.71,A -85,B 0,C 180,E1 -18316.34,E2 -18316.34} C_VEL
LIN {X 0,Y 263.157,Z 236.701,A -85,B 0,C 180,E1 -18320.136,E2 -18320.136} C_VEL
LIN {X 0,Y 263.171,Z 236.705,A -85,B 0,C 180,E1 -18324.019,E2 -18324.019} C_VEL
LIN {X 0,Y 263.125,Z 236.709,A -85,B 0,C 180,E1 -18327.71,E2 -18327.71} C_VEL
LIN {X 0,Y 263.192,Z 236.695,A -85,B 0,C 180,E1 -18331.782,E2 -18331.782} C_VEL
LIN {X 0,Y 263.191,Z 236.698,A -85,B 0,C 180,E1 -18335.212,E2 -18335.212} C_VEL
LIN {X 0,Y 263.226,Z 236.688,A -85,B 0,C 180,E1 -18339.69,E2 -18339.69} C_VEL
LIN {X 0,Y 263.311,Z 236.674,A -85,B 0,C 180,E1 -18344.519,E2 -18344.519} C_VEL
LIN {X 0,Y 263.32,Z 236.675,A -85,B 0,C 180,E1 -18349.232,E2 -18349.232} C_VEL
LIN {X 0,Y 263.357,Z 236.671,A -85,B 0,C 180,E1 -18349.854,E2 -18349.854} C_VEL
LIN {X 0,Y 263.091,Z 236.711,A -85,B 0,C 180,E1 -18350.708,E2 -18350.708} C_VEL
LIN {X 0,Y 261.754,Z 236.88,A -85,B 0,C 180,E1 -18351.969,E2 -18351.969} C_VEL
LIN {X 0,Y 257.417,Z 237.415,A -85,B 0,C 180,E1 -18354.905,E2 -18354.905} C_VEL
LIN {X 0,Y 256.468,Z 237.538,A -85,B 0,C 180,E1 -18356.219,E2 -18356.219} C_VEL
LIN {X 0,Y 256.444,Z 237.537,A -85,B 0,C 180,E1 -18356.664,E2 -18356.664} C_VEL
LIN {X 0,Y 256.695,Z 237.497,A -85,B 0,C 180,E1 -18358.431,E2 -18358.431} C_VEL
LIN {X 0,Y 256.69,Z 237.506,A -85,B 0,C 180,E1 -18361.569,E2 -18361.569} C_VEL
LIN {X 0,Y 256.438,Z 237.539,A -85,B 0,C 180,E1 -18366.294,E2 -18366.294} C_VEL
LIN {X 0,Y 256.387,Z 237.547,A -85,B 0,C 180,E1 -18369.466,E2 -18369.466} C_VEL
LIN {X 0,Y 256.216,Z 237.567,A -85,B 0,C 180,E1 -18374.292,E2 -18374.292} C_VEL
LIN {X 0,Y 256.148,Z 237.568,A -85,B 0,C 180,E1 -18377.566,E2 -18377.566} C_VEL
LIN {X 0,Y 256.107,Z 237.572,A -85,B 0,C 180,E1 -18381.096,E2 -18381.096} C_VEL
LIN {X 0,Y 256.067,Z 237.579,A -85,B 0,C 180,E1 -18385.085,E2 -18385.085} C_VEL
LIN {X 0,Y 256.066,Z 237.585,A -85,B 0,C 180,E1 -18388.569,E2 -18388.569} C_VEL
LIN {X 0,Y 256.054,Z 237.59,A -85,B 0,C 180,E1 -18391.697,E2 -18391.697} C_VEL
LIN {X 0,Y 256.071,Z 237.587,A -85,B 0,C 180,E1 -18395.195,E2 -18395.195} C_VEL
LIN {X 0,Y 256.063,Z 237.559,A -85,B 0,C 180,E1 -18399.144,E2 -18399.144} C_VEL
LIN {X 0,Y 256.042,Z 237.588,A -85,B 0,C 180,E1 -18403.331,E2 -18403.331} C_VEL
LIN {X 0,Y 256.072,Z 237.658,A -85,B 0,C 180,E1 -18406.676,E2 -18406.676} C_VEL
LIN {X 0,Y 258.757,Z 246.98,A -85,B 0,C 180,E1 -18410.961,E2 -18410.961} C_VEL
LIN {X 0,Y 260.955,Z 255.284,A -85,B 0,C 180,E1 -18414.372,E2 -18414.372} C_VEL
LIN {X 0,Y 268.416,Z 270.089,A -85,B 0,C 180,E1 -18416.182,E2 -18416.182} C_VEL
LIN {X 0,Y 274.476,Z 283.162,A -85,B 0,C 180,E1 -18417.58,E2 -18417.58} C_VEL
LIN {X 0,Y 277.592,Z 300.493,A -85,B 0,C 180,E1 -18418.598,E2 -18418.598} C_VEL
LIN {X 0,Y 279.172,Z 312.539,A -85,B 0,C 180,E1 -18419.201,E2 -18419.201} C_VEL
LIN {X 0,Y 277.042,Z 365.55,A -85,B 0,C 180,E1 -18420.588,E2 -18420.588} C_VEL
LIN {X 0,Y 275.595,Z 379.584,A -85,B 0,C 180,E1 -18421.227,E2 -18421.227} C_VEL
LIN {X 0,Y 273.789,Z 391.793,A -85,B 0,C 180,E1 -18422.065,E2 -18422.065} C_VEL
LIN {X 0,Y 271.396,Z 404.346,A -85,B 0,C 180,E1 -18423.26,E2 -18423.26} C_VEL
LIN {X 0,Y 268.882,Z 415.544,A -85,B 0,C 180,E1 -18424.658,E2 -18424.658} C_VEL
LIN {X 0,Y 266.257,Z 425.664,A -85,B 0,C 180,E1 -18426.263,E2 -18426.263} C_VEL
LIN {X 0,Y 263.741,Z 434.798,A -85,B 0,C 180,E1 -18428.095,E2 -18428.095} C_VEL
LIN {X 0,Y 261.039,Z 443.658,A -85,B 0,C 180,E1 -18430.313,E2 -18430.313} C_VEL
LIN {X 0,Y 258.924,Z 450.935,A -85,B 0,C 180,E1 -18432.627,E2 -18432.627} C_VEL
LIN {X 0,Y 257.135,Z 456.726,A -85,B 0,C 180,E1 -18434.949,E2 -18434.949} C_VEL
LIN {X 0,Y 255.697,Z 461.313,A -85,B 0,C 180,E1 -18437.296,E2 -18437.296} C_VEL
LIN {X 0,Y 254.819,Z 464.829,A -85,B 0,C 180,E1 -18439.671,E2 -18439.671} C_VEL
LIN {X 0,Y 254.263,Z 467.359,A -85,B 0,C 180,E1 -18442.054,E2 -18442.054} C_VEL
LIN {X 0,Y 254.022,Z 469.186,A -85,B 0,C 180,E1 -18444.879,E2 -18444.879} C_VEL
LIN {X 0,Y 254.075,Z 469.685,A -85,B 0,C 180,E1 -18446.826,E2 -18446.826} C_VEL
LIN {X 0,Y 254.122,Z 469.677,A -85,B 0,C 180,E1 -18448.412,E2 -18448.412} C_VEL
LIN {X 0,Y 254.173,Z 469.272,A -85,B 0,C 180,E1 -18449.997,E2 -18449.997} C_VEL
LIN {X 0,Y 254.153,Z 468.421,A -85,B 0,C 180,E1 -18451.581,E2 -18451.581} C_VEL
LIN {X 0,Y 254.13,Z 467.162,A -85,B 0,C 180,E1 -18453.167,E2 -18453.167} C_VEL
LIN {X 0,Y 254.09,Z 464.819,A -85,B 0,C 180,E1 -18455.288,E2 -18455.288} C_VEL
LIN {X 0,Y 254.304,Z 460.723,A -85,B 0,C 180,E1 -18457.939,E2 -18457.939} C_VEL
LIN {X 0,Y 254.693,Z 455.835,A -85,B 0,C 180,E1 -18460.329,E2 -18460.329} C_VEL
LIN {X 0,Y 255.399,Z 449.654,A -85,B 0,C 180,E1 -18462.713,E2 -18462.713} C_VEL
LIN {X 0,Y 256.589,Z 441.969,A -85,B 0,C 180,E1 -18465.078,E2 -18465.078} C_VEL
LIN {X 0,Y 257.742,Z 434.076,A -85,B 0,C 180,E1 -18467.04,E2 -18467.04} C_VEL
LIN {X 0,Y 259.305,Z 424.435,A -85,B 0,C 180,E1 -18468.975,E2 -18468.975} C_VEL
LIN {X 0,Y 260.859,Z 413.716,A -85,B 0,C 180,E1 -18470.703,E2 -18470.703} C_VEL
LIN {X 0,Y 262.554,Z 401.702,A -85,B 0,C 180,E1 -18472.21,E2 -18472.21} C_VEL
LIN {X 0,Y 263.993,Z 389.95,A -85,B 0,C 180,E1 -18473.323,E2 -18473.323} C_VEL
LIN {X 0,Y 265.286,Z 376.613,A -85,B 0,C 180,E1 -18474.239,E2 -18474.239} C_VEL
LIN {X 0,Y 266.069,Z 364.384,A -85,B 0,C 180,E1 -18474.786,E2 -18474.786} C_VEL
LIN {X 0,Y 267.464,Z 306.111,A -85,B 0,C 180,E1 -18476.354,E2 -18476.354} C_VEL
LIN {X 0,Y 262.83,Z 268.079,A -85,B 0,C 180,E1 -18477.871,E2 -18477.871} C_VEL
LIN {X 0,Y 261.552,Z 260.798,A -85,B 0,C 180,E1 -18478.207,E2 -18478.207} C_VEL
LIN {X 0,Y 260.098,Z 256.465,A -85,B 0,C 180,E1 -18478.512,E2 -18478.512} C_VEL
LIN {X 0,Y 257.817,Z 245.247,A -85,B 0,C 180,E1 -18482.323,E2 -18482.323} C_VEL
LIN {X 0,Y 256.108,Z 237.586,A -85,B 0,C 180,E1 -18485.091,E2 -18485.091} C_VEL
LIN {X 0,Y 256.053,Z 237.59,A -85,B 0,C 180,E1 -18489.137,E2 -18489.137} C_VEL
LIN {X 0,Y 256.044,Z 237.591,A -85,B 0,C 180,E1 -18493.321,E2 -18493.321} C_VEL
LIN {X 0,Y 256.096,Z 237.586,A -85,B 0,C 180,E1 -18497.802,E2 -18497.802} C_VEL
LIN {X 0,Y 256.081,Z 237.585,A -85,B 0,C 180,E1 -18500.86,E2 -18500.86} C_VEL
LIN {X 0,Y 256.061,Z 237.588,A -85,B 0,C 180,E1 -18504.804,E2 -18504.804} C_VEL
LIN {X 0,Y 256.061,Z 237.588,A -85,B 0,C 180,E1 -18508.568,E2 -18508.568} C_VEL
LIN {X 0,Y 256.11,Z 237.581,A -85,B 0,C 180,E1 -18512.193,E2 -18512.193} C_VEL
LIN {X 0,Y 256.153,Z 237.578,A -85,B 0,C 180,E1 -18515.698,E2 -18515.698} C_VEL
LIN {X 0,Y 256.205,Z 237.571,A -85,B 0,C 180,E1 -18519.108,E2 -18519.108} C_VEL
LIN {X 0,Y 256.227,Z 237.566,A -85,B 0,C 180,E1 -18524.081,E2 -18524.081} C_VEL
LIN {X 0,Y 256.25,Z 237.563,A -85,B 0,C 180,E1 -18527.326,E2 -18527.326} C_VEL
LIN {X 0,Y 256.482,Z 237.531,A -85,B 0,C 180,E1 -18532.125,E2 -18532.125} C_VEL
LIN {X 0,Y 256.456,Z 237.54,A -85,B 0,C 180,E1 -18536.858,E2 -18536.858} C_VEL
LIN {X 0,Y 256.714,Z 237.495,A -85,B 0,C 180,E1 -18540,E2 -18540} C_VEL
LIN {X 0,Y 256.448,Z 237.524,A -85,B 0,C 180,E1 -18543.142,E2 -18543.142} C_VEL
LIN {X 0,Y 256.47,Z 237.535,A -85,B 0,C 180,E1 -18547.875,E2 -18547.875} C_VEL
LIN {X 0,Y 256.219,Z 237.557,A -85,B 0,C 180,E1 -18552.676,E2 -18552.676} C_VEL
LIN {X 0,Y 256.179,Z 237.561,A -85,B 0,C 180,E1 -18556.252,E2 -18556.252} C_VEL
LIN {X 0,Y 256.086,Z 237.584,A -85,B 0,C 180,E1 -18561.101,E2 -18561.101} C_VEL
LIN {X 0,Y 256.137,Z 237.578,A -85,B 0,C 180,E1 -18565.132,E2 -18565.132} C_VEL
LIN {X 0,Y 256.073,Z 237.583,A -85,B 0,C 180,E1 -18569.605,E2 -18569.605} C_VEL
LIN {X 0,Y 256.039,Z 237.588,A -85,B 0,C 180,E1 -18573.297,E2 -18573.297} C_VEL
LIN {X 0,Y 256.109,Z 237.581,A -85,B 0,C 180,E1 -18577.281,E2 -18577.281} C_VEL
LIN {X 0,Y 256.076,Z 237.584,A -85,B 0,C 180,E1 -18581.2,E2 -18581.2} C_VEL
LIN {X 0,Y 256.044,Z 237.579,A -85,B 0,C 180,E1 -18585.534,E2 -18585.534} C_VEL
LIN {X 0,Y 256.035,Z 237.589,A -85,B 0,C 180,E1 -18588.802,E2 -18588.802} C_VEL
LIN {X 0,Y 256.113,Z 237.572,A -85,B 0,C 180,E1 -18592.872,E2 -18592.872} C_VEL
LIN {X 0,Y 256.054,Z 237.587,A -85,B 0,C 180,E1 -18596.712,E2 -18596.712} C_VEL
LIN {X 0,Y 256.093,Z 237.585,A -85,B 0,C 180,E1 -18600.404,E2 -18600.404} C_VEL
LIN {X 0,Y 256.163,Z 237.572,A -85,B 0,C 180,E1 -18604.875,E2 -18604.875} C_VEL
LIN {X 0,Y 256.142,Z 237.576,A -85,B 0,C 180,E1 -18609.108,E2 -18609.108} C_VEL
LIN {X 0,Y 256.157,Z 237.643,A -85,B 0,C 180,E1 -18612.285,E2 -18612.285} C_VEL
LIN {X 0,Y 257.296,Z 240.601,A -85,B 0,C 180,E1 -18612.491,E2 -18612.491} C_VEL
LIN {X 0,Y 263.068,Z 253.383,A -85,B 0,C 180,E1 -18613.442,E2 -18613.442} C_VEL
LIN {X 0,Y 268.567,Z 269.421,A -85,B 0,C 180,E1 -18614.416,E2 -18614.416} C_VEL
LIN {X 0,Y 266.343,Z 341.705,A -85,B 0,C 180,E1 -18616.315,E2 -18616.315} C_VEL
LIN {X 0,Y 265.509,Z 354.547,A -85,B 0,C 180,E1 -18616.904,E2 -18616.904} C_VEL
LIN {X 0,Y 264.721,Z 366.347,A -85,B 0,C 180,E1 -18617.742,E2 -18617.742} C_VEL
LIN {X 0,Y 263.651,Z 378.063,A -85,B 0,C 180,E1 -18618.861,E2 -18618.861} C_VEL
LIN {X 0,Y 262.244,Z 388.786,A -85,B 0,C 180,E1 -18620.167,E2 -18620.167} C_VEL
LIN {X 0,Y 260.824,Z 398.644,A -85,B 0,C 180,E1 -18621.676,E2 -18621.676} C_VEL
LIN {X 0,Y 259.377,Z 407.722,A -85,B 0,C 180,E1 -18623.391,E2 -18623.391} C_VEL
LIN {X 0,Y 258.071,Z 416.025,A -85,B 0,C 180,E1 -18625.317,E2 -18625.317} C_VEL
LIN {X 0,Y 256.768,Z 424.156,A -85,B 0,C 180,E1 -18627.65,E2 -18627.65} C_VEL
LIN {X 0,Y 255.71,Z 430.711,A -85,B 0,C 180,E1 -18630.003,E2 -18630.003} C_VEL
LIN {X 0,Y 255.066,Z 435.923,A -85,B 0,C 180,E1 -18632.371,E2 -18632.371} C_VEL
LIN {X 0,Y 254.615,Z 439.983,A -85,B 0,C 180,E1 -18634.752,E2 -18634.752} C_VEL
LIN {X 0,Y 254.371,Z 442.101,A -85,B 0,C 180,E1 -18636.347,E2 -18636.347} C_VEL
LIN {X 0,Y 254.128,Z 443.786,A -85,B 0,C 180,E1 -18637.95,E2 -18637.95} C_VEL
LIN {X 0,Y 254.014,Z 445.066,A -85,B 0,C 180,E1 -18639.558,E2 -18639.558} C_VEL
LIN {X 0,Y 253.967,Z 445.939,A -85,B 0,C 180,E1 -18641.171,E2 -18641.171} C_VEL
LIN {X 0,Y 254.11,Z 446.367,A -85,B 0,C 180,E1 -18642.785,E2 -18642.785} C_VEL
LIN {X 0,Y 254.357,Z 446.378,A -85,B 0,C 180,E1 -18644.744,E2 -18644.744} C_VEL
LIN {X 0,Y 254.895,Z 445.286,A -85,B 0,C 180,E1 -18647.657,E2 -18647.657} C_VEL
LIN {X 0,Y 255.413,Z 444.066,A -85,B 0,C 180,E1 -18649.282,E2 -18649.282} C_VEL
LIN {X 0,Y 256.185,Z 442.176,A -85,B 0,C 180,E1 -18651.134,E2 -18651.134} C_VEL
LIN {X 0,Y 257.309,Z 439.104,A -85,B 0,C 180,E1 -18653.332,E2 -18653.332} C_VEL
LIN {X 0,Y 258.904,Z 434.644,A -85,B 0,C 180,E1 -18655.743,E2 -18655.743} C_VEL
LIN {X 0,Y 260.895,Z 428.915,A -85,B 0,C 180,E1 -18658.127,E2 -18658.127} C_VEL
LIN {X 0,Y 263.215,Z 421.642,A -85,B 0,C 180,E1 -18660.485,E2 -18660.485} C_VEL
LIN {X 0,Y 265.953,Z 412.519,A -85,B 0,C 180,E1 -18662.801,E2 -18662.801} C_VEL
LIN {X 0,Y 268.461,Z 403.043,A -85,B 0,C 180,E1 -18664.707,E2 -18664.707} C_VEL
LIN {X 0,Y 271.066,Z 392.422,A -85,B 0,C 180,E1 -18666.373,E2 -18666.373} C_VEL
LIN {X 0,Y 273.374,Z 380.477,A -85,B 0,C 180,E1 -18667.863,E2 -18667.863} C_VEL
LIN {X 0,Y 275.177,Z 368.769,A -85,B 0,C 180,E1 -18668.97,E2 -18668.97} C_VEL
LIN {X 0,Y 276.791,Z 355.587,A -85,B 0,C 180,E1 -18669.863,E2 -18669.863} C_VEL
LIN {X 0,Y 277.855,Z 342.906,A -85,B 0,C 180,E1 -18670.431,E2 -18670.431} C_VEL
LIN {X 0,Y 280.255,Z 282.153,A -85,B 0,C 180,E1 -18671.999,E2 -18671.999} C_VEL
LIN {X 0,Y 272.971,Z 266.672,A -85,B 0,C 180,E1 -18673.604,E2 -18673.604} C_VEL
LIN {X 0,Y 265.774,Z 253.41,A -85,B 0,C 180,E1 -18675.249,E2 -18675.249} C_VEL
LIN {X 0,Y 260.269,Z 245.072,A -85,B 0,C 180,E1 -18676.533,E2 -18676.533} C_VEL
LIN {X 0,Y 258.301,Z 241.817,A -85,B 0,C 180,E1 -18677.022,E2 -18677.022} C_VEL
LIN {X 0,Y 256.63,Z 239.434,A -85,B 0,C 180,E1 -18677.433,E2 -18677.433} C_VEL
LIN {X 0,Y 256.147,Z 237.577,A -85,B 0,C 180,E1 -18677.65,E2 -18677.65} C_VEL
LIN {X 0,Y 256.104,Z 237.584,A -85,B 0,C 180,E1 -18680.863,E2 -18680.863} C_VEL
LIN {X 0,Y 256.083,Z 237.584,A -85,B 0,C 180,E1 -18684.807,E2 -18684.807} C_VEL
LIN {X 0,Y 256.084,Z 237.579,A -85,B 0,C 180,E1 -18688.571,E2 -18688.571} C_VEL
LIN {X 0,Y 256.132,Z 237.571,A -85,B 0,C 180,E1 -18692.195,E2 -18692.195} C_VEL
LIN {X 0,Y 256.131,Z 237.572,A -85,B 0,C 180,E1 -18695.695,E2 -18695.695} C_VEL
LIN {X 0,Y 256.136,Z 237.577,A -85,B 0,C 180,E1 -18699.102,E2 -18699.102} C_VEL
LIN {X 0,Y 256.247,Z 237.556,A -85,B 0,C 180,E1 -18704.081,E2 -18704.081} C_VEL
LIN {X 0,Y 256.266,Z 237.553,A -85,B 0,C 180,E1 -18708.932,E2 -18708.932} C_VEL
LIN {X 0,Y 256.497,Z 237.532,A -85,B 0,C 180,E1 -18712.126,E2 -18712.126} C_VEL
LIN {X 0,Y 256.444,Z 237.537,A -85,B 0,C 180,E1 -18716.664,E2 -18716.664} C_VEL
LIN {X 0,Y 255.927,Z 237.606,A -85,B 0,C 180,E1 -18717.977,E2 -18717.977} C_VEL
LIN {X 0,Y 254.409,Z 237.795,A -85,B 0,C 180,E1 -18719.268,E2 -18719.268} C_VEL
LIN {X 0,Y 250.617,Z 238.261,A -85,B 0,C 180,E1 -18721.86,E2 -18721.86} C_VEL
LIN {X 0,Y 249.462,Z 238.399,A -85,B 0,C 180,E1 -18723.212,E2 -18723.212} C_VEL
LIN {X 0,Y 249.333,Z 238.415,A -85,B 0,C 180,E1 -18723.672,E2 -18723.672} C_VEL
LIN {X 0,Y 249.409,Z 238.412,A -85,B 0,C 180,E1 -18726.472,E2 -18726.472} C_VEL
LIN {X 0,Y 249.321,Z 238.427,A -85,B 0,C 180,E1 -18729.737,E2 -18729.737} C_VEL
LIN {X 0,Y 249.157,Z 238.449,A -85,B 0,C 180,E1 -18734.706,E2 -18734.706} C_VEL
LIN {X 0,Y 249.081,Z 238.452,A -85,B 0,C 180,E1 -18738.082,E2 -18738.082} C_VEL
LIN {X 0,Y 249.032,Z 238.453,A -85,B 0,C 180,E1 -18741.523,E2 -18741.523} C_VEL
LIN {X 0,Y 249.029,Z 238.454,A -85,B 0,C 180,E1 -18745.437,E2 -18745.437} C_VEL
LIN {X 0,Y 249.014,Z 238.46,A -85,B 0,C 180,E1 -18748.968,E2 -18748.968} C_VEL
LIN {X 0,Y 248.988,Z 238.466,A -85,B 0,C 180,E1 -18752.432,E2 -18752.432} C_VEL
LIN {X 0,Y 249.008,Z 238.458,A -85,B 0,C 180,E1 -18756.349,E2 -18756.349} C_VEL
LIN {X 0,Y 248.985,Z 238.457,A -85,B 0,C 180,E1 -18760.482,E2 -18760.482} C_VEL
LIN {X 0,Y 248.993,Z 238.465,A -85,B 0,C 180,E1 -18762.79,E2 -18762.79} C_VEL
LIN {X 0,Y 249.013,Z 238.555,A -85,B 0,C 180,E1 -18765.455,E2 -18765.455} C_VEL
LIN {X 0,Y 251.515,Z 247.096,A -85,B 0,C 180,E1 -18769.603,E2 -18769.603} C_VEL
LIN {X 0,Y 253.573,Z 254.686,A -85,B 0,C 180,E1 -18772.944,E2 -18772.944} C_VEL
LIN {X 0,Y 256.072,Z 259.303,A -85,B 0,C 180,E1 -18773.602,E2 -18773.602} C_VEL
LIN {X 0,Y 263.267,Z 273.457,A -85,B 0,C 180,E1 -18775.419,E2 -18775.419} C_VEL
LIN {X 0,Y 269.12,Z 286.302,A -85,B 0,C 180,E1 -18776.837,E2 -18776.837} C_VEL
LIN {X 0,Y 272.933,Z 309.362,A -85,B 0,C 180,E1 -18778.184,E2 -18778.184} C_VEL
LIN {X 0,Y 273.321,Z 314.013,A -85,B 0,C 180,E1 -18778.391,E2 -18778.391} C_VEL
LIN {X 0,Y 271.136,Z 365.445,A -85,B 0,C 180,E1 -18779.761,E2 -18779.761} C_VEL
LIN {X 0,Y 269.743,Z 378.83,A -85,B 0,C 180,E1 -18780.382,E2 -18780.382} C_VEL
LIN {X 0,Y 267.757,Z 391.686,A -85,B 0,C 180,E1 -18781.271,E2 -18781.271} C_VEL
LIN {X 0,Y 265.464,Z 403.403,A -85,B 0,C 180,E1 -18782.399,E2 -18782.399} C_VEL
